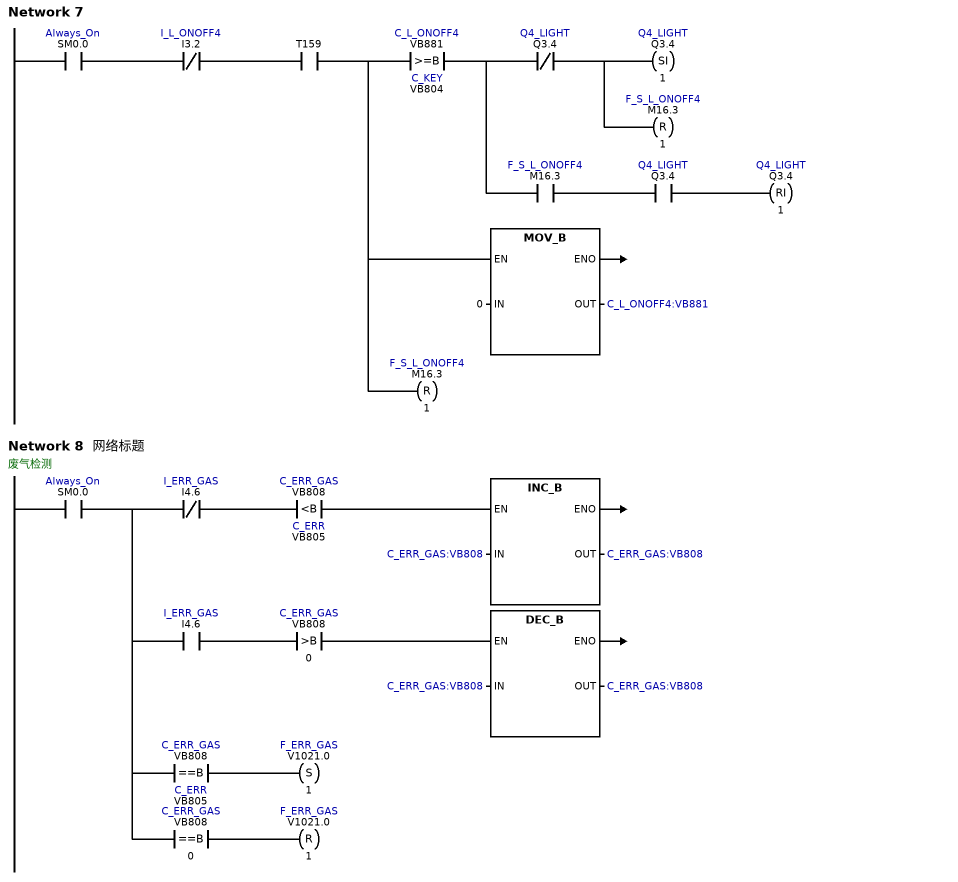
[picture p24: SBR3 networks 7-8]
Network 7
LD     Always_On:SM0.0
AN     I_L_ONOFF4:I3.2
A      T159
LPS
AB>=   C_L_ONOFF4:VB881, C_KEY:VB804
LPS
AN     Q4_LIGHT:Q3.4
SI     Q4_LIGHT:Q3.4, 1
R      F_S_L_ONOFF4:M16.3, 1
LPP
A      F_S_L_ONOFF4:M16.3
A      Q4_LIGHT:Q3.4
RI     Q4_LIGHT:Q3.4, 1
LPP
MOVB   0, C_L_ONOFF4:VB881
R      F_S_L_ONOFF4:M16.3, 1
Network 8 // 网络标题
// 废气检测
LD     Always_On:SM0.0
LPS
AN     I_ERR_GAS:I4.6
AB<    C_ERR_GAS:VB808, C_ERR:VB805
INCB   C_ERR_GAS:VB808
LRD
A      I_ERR_GAS:I4.6
AB>    C_ERR_GAS:VB808, 0
DECB   C_ERR_GAS:VB808
LRD
AB=    C_ERR_GAS:VB808, C_ERR:VB805
S      F_ERR_GAS:V1021.0, 1
LPP
AB=    C_ERR_GAS:VB808, 0
R      F_ERR_GAS:V1021.0, 1
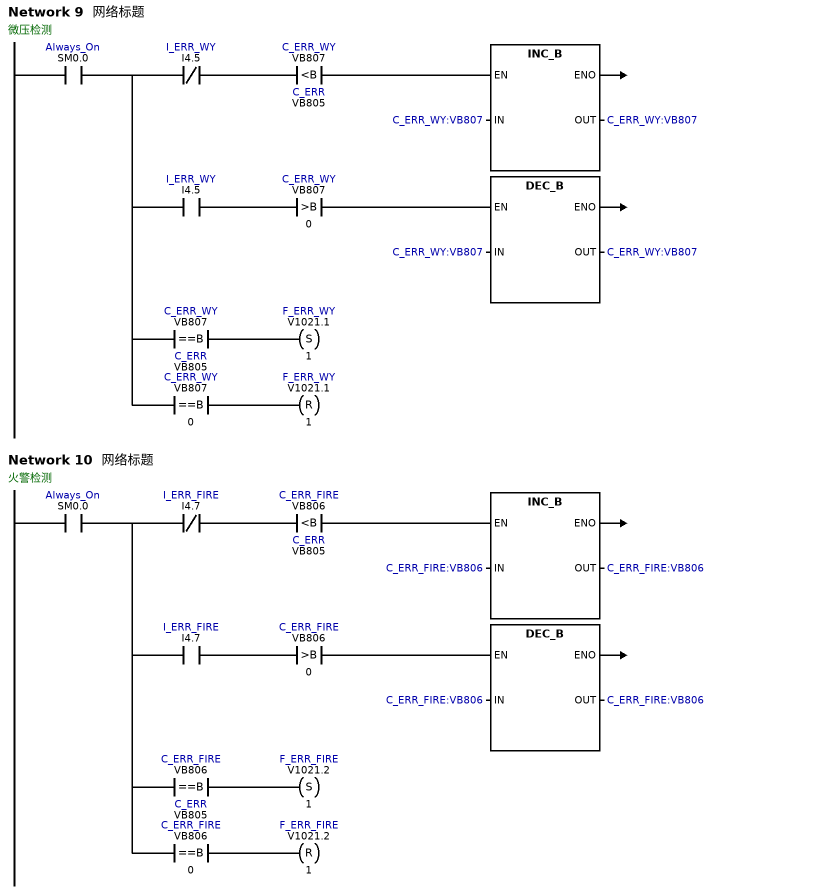
Network 9 // 网络标题
// 微压检测
LD     Always_On:SM0.0
LPS
AN     I_ERR_WY:I4.5
AB<    C_ERR_WY:VB807, C_ERR:VB805
INCB   C_ERR_WY:VB807
LRD
A      I_ERR_WY:I4.5
AB>    C_ERR_WY:VB807, 0
DECB   C_ERR_WY:VB807
LRD
AB=    C_ERR_WY:VB807, C_ERR:VB805
S      F_ERR_WY:V1021.1, 1
LPP
AB=    C_ERR_WY:VB807, 0
R      F_ERR_WY:V1021.1, 1
Network 10 // 网络标题
// 火警检测
LD     Always_On:SM0.0
LPS
AN     I_ERR_FIRE:I4.7
AB<    C_ERR_FIRE:VB806, C_ERR:VB805
INCB   C_ERR_FIRE:VB806
LRD
A      I_ERR_FIRE:I4.7
AB>    C_ERR_FIRE:VB806, 0
DECB   C_ERR_FIRE:VB806
LRD
AB=    C_ERR_FIRE:VB806, C_ERR:VB805
S      F_ERR_FIRE:V1021.2, 1
LPP
AB=    C_ERR_FIRE:VB806, 0
R      F_ERR_FIRE:V1021.2, 1
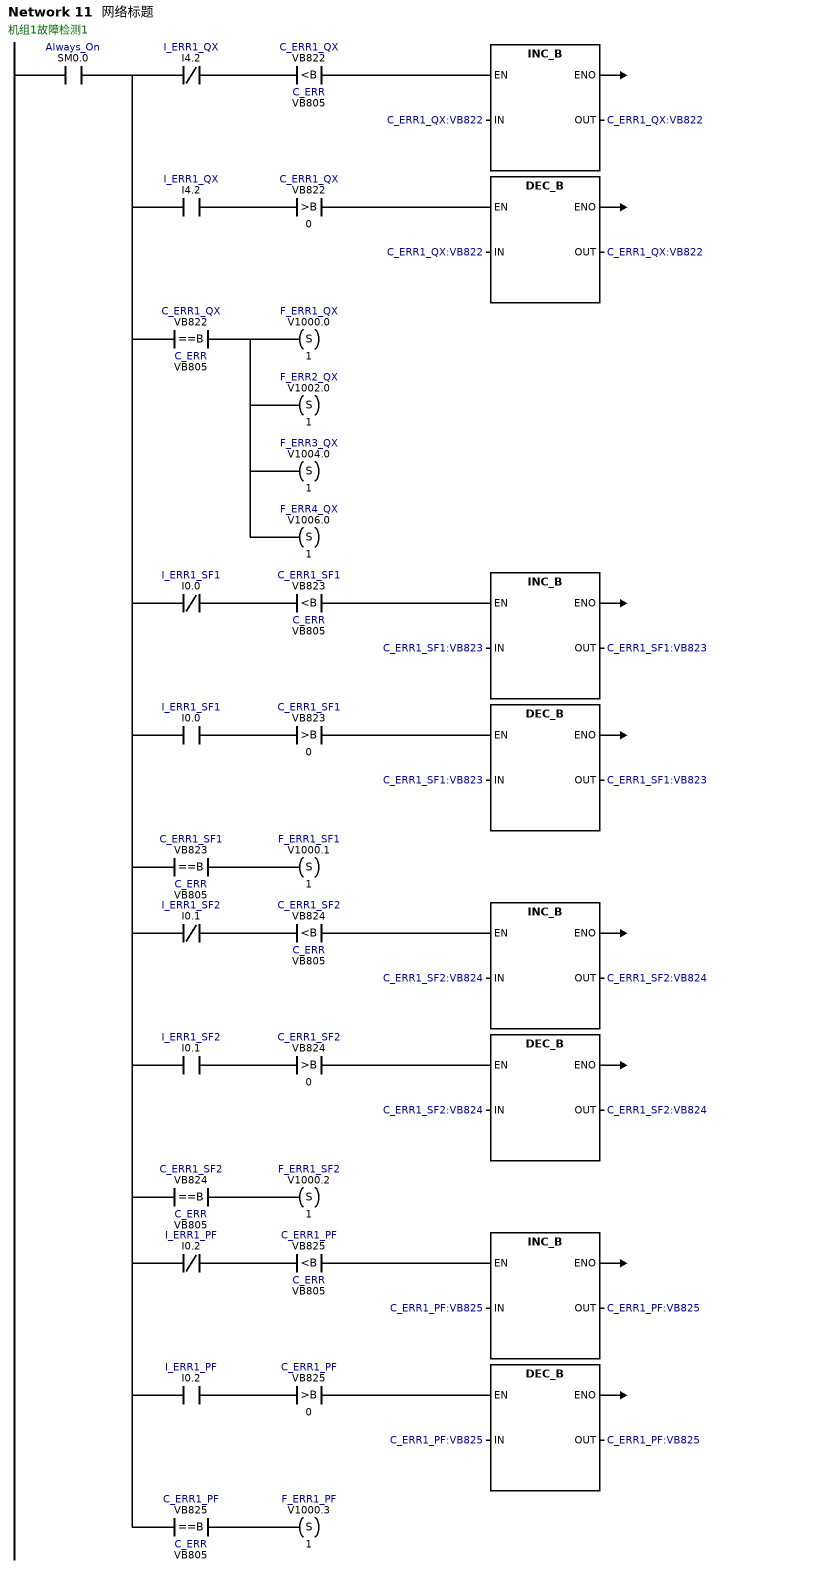
Network 11 // 网络标题
// 机组1故障检测1
LD     Always_On:SM0.0
LPS
AN     I_ERR1_QX:I4.2
AB<    C_ERR1_QX:VB822, C_ERR:VB805
INCB   C_ERR1_QX:VB822
LRD
A      I_ERR1_QX:I4.2
AB>    C_ERR1_QX:VB822, 0
DECB   C_ERR1_QX:VB822
LRD
AB=    C_ERR1_QX:VB822, C_ERR:VB805
S      F_ERR1_QX:V1000.0, 1
S      F_ERR2_QX:V1002.0, 1
S      F_ERR3_QX:V1004.0, 1
S      F_ERR4_QX:V1006.0, 1
LPP
LPS
AN     I_ERR1_SF1:I0.0
AB<    C_ERR1_SF1:VB823, C_ERR:VB805
INCB   C_ERR1_SF1:VB823
LRD
A      I_ERR1_SF1:I0.0
AB>    C_ERR1_SF1:VB823, 0
DECB   C_ERR1_SF1:VB823
LRD
AB=    C_ERR1_SF1:VB823, C_ERR:VB805
S      F_ERR1_SF1:V1000.1, 1
LRD
AN     I_ERR1_SF2:I0.1
AB<    C_ERR1_SF2:VB824, C_ERR:VB805
INCB   C_ERR1_SF2:VB824
LRD
A      I_ERR1_SF2:I0.1
AB>    C_ERR1_SF2:VB824, 0
DECB   C_ERR1_SF2:VB824
LRD
AB=    C_ERR1_SF2:VB824, C_ERR:VB805
S      F_ERR1_SF2:V1000.2, 1
LRD
AN     I_ERR1_PF:I0.2
AB<    C_ERR1_PF:VB825, C_ERR:VB805
INCB   C_ERR1_PF:VB825
LRD
A      I_ERR1_PF:I0.2
AB>    C_ERR1_PF:VB825, 0
DECB   C_ERR1_PF:VB825
LPP
AB=    C_ERR1_PF:VB825, C_ERR:VB805
S      F_ERR1_PF:V1000.3, 1
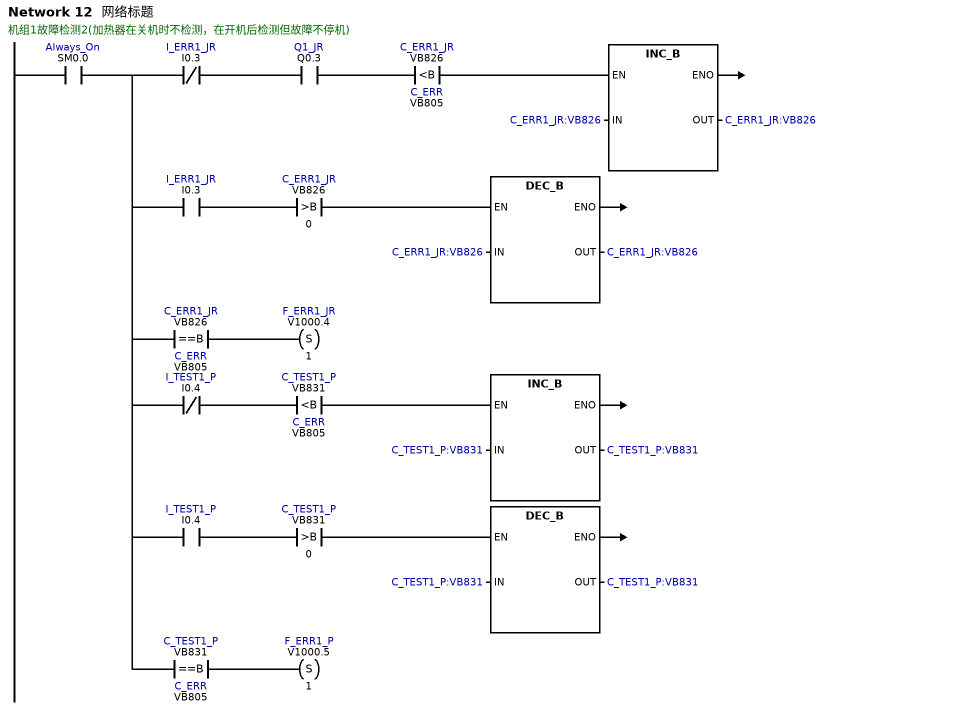
Network 12 // 网络标题
// 机组1故障检测2(加热器在关机时不检测，在开机后检测但故障不停机)
LD     Always_On:SM0.0
LPS
AN     I_ERR1_JR:I0.3
A      Q1_JR:Q0.3
AB<    C_ERR1_JR:VB826, C_ERR:VB805
INCB   C_ERR1_JR:VB826
LRD
A      I_ERR1_JR:I0.3
AB>    C_ERR1_JR:VB826, 0
DECB   C_ERR1_JR:VB826
LRD
AB=    C_ERR1_JR:VB826, C_ERR:VB805
S      F_ERR1_JR:V1000.4, 1
LRD
AN     I_TEST1_P:I0.4
AB<    C_TEST1_P:VB831, C_ERR:VB805
INCB   C_TEST1_P:VB831
LRD
A      I_TEST1_P:I0.4
AB>    C_TEST1_P:VB831, 0
DECB   C_TEST1_P:VB831
LPP
AB=    C_TEST1_P:VB831, C_ERR:VB805
S      F_ERR1_P:V1000.5, 1
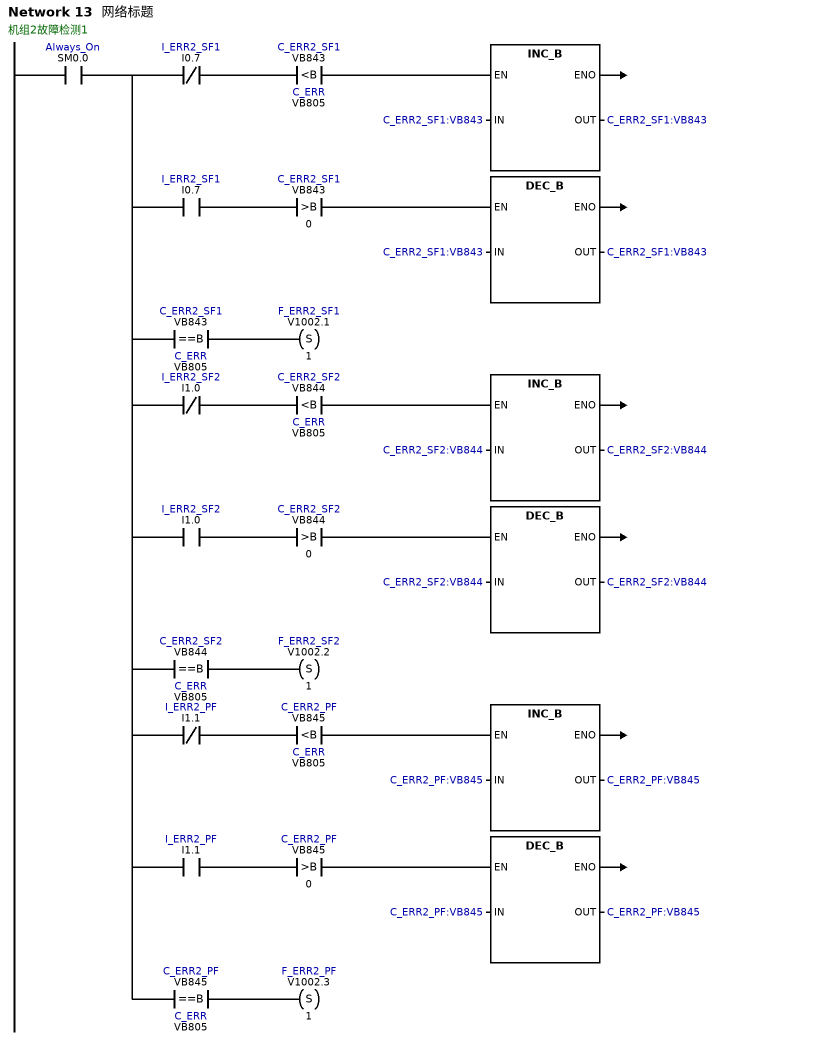
Network 13 // 网络标题
// 机组2故障检测1
LD     Always_On:SM0.0
LPS
AN     I_ERR2_SF1:I0.7
AB<    C_ERR2_SF1:VB843, C_ERR:VB805
INCB   C_ERR2_SF1:VB843
LRD
A      I_ERR2_SF1:I0.7
AB>    C_ERR2_SF1:VB843, 0
DECB   C_ERR2_SF1:VB843
LRD
AB=    C_ERR2_SF1:VB843, C_ERR:VB805
S      F_ERR2_SF1:V1002.1, 1
LRD
AN     I_ERR2_SF2:I1.0
AB<    C_ERR2_SF2:VB844, C_ERR:VB805
INCB   C_ERR2_SF2:VB844
LRD
A      I_ERR2_SF2:I1.0
AB>    C_ERR2_SF2:VB844, 0
DECB   C_ERR2_SF2:VB844
LRD
AB=    C_ERR2_SF2:VB844, C_ERR:VB805
S      F_ERR2_SF2:V1002.2, 1
LRD
AN     I_ERR2_PF:I1.1
AB<    C_ERR2_PF:VB845, C_ERR:VB805
INCB   C_ERR2_PF:VB845
LRD
A      I_ERR2_PF:I1.1
AB>    C_ERR2_PF:VB845, 0
DECB   C_ERR2_PF:VB845
LPP
AB=    C_ERR2_PF:VB845, C_ERR:VB805
S      F_ERR2_PF:V1002.3, 1
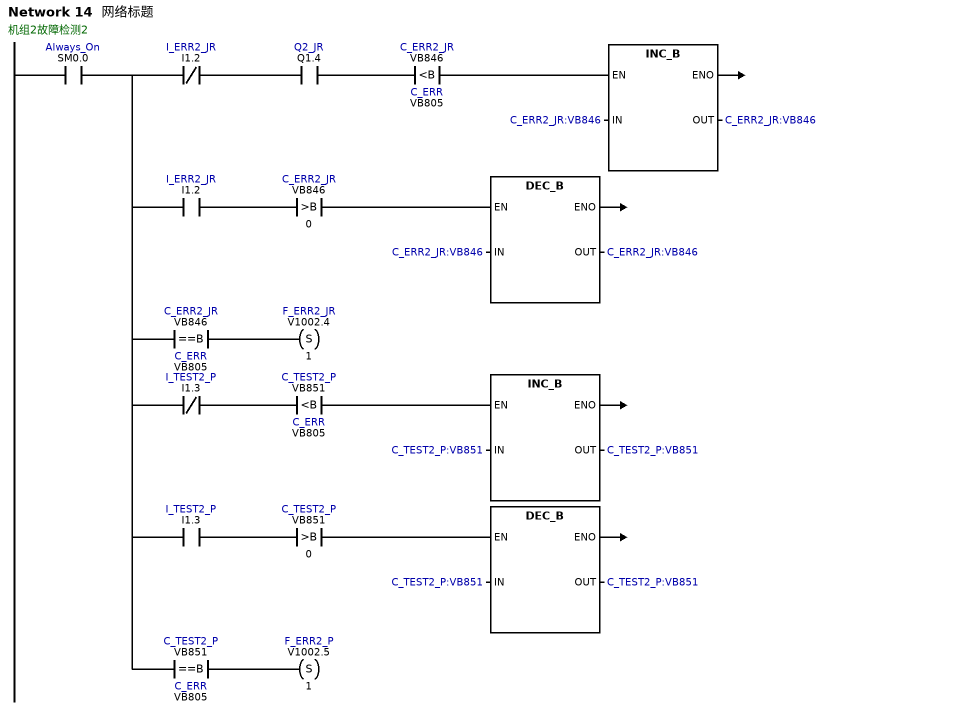
Network 14 // 网络标题
// 机组2故障检测2
LD     Always_On:SM0.0
LPS
AN     I_ERR2_JR:I1.2
A      Q2_JR:Q1.4
AB<    C_ERR2_JR:VB846, C_ERR:VB805
INCB   C_ERR2_JR:VB846
LRD
A      I_ERR2_JR:I1.2
AB>    C_ERR2_JR:VB846, 0
DECB   C_ERR2_JR:VB846
LRD
AB=    C_ERR2_JR:VB846, C_ERR:VB805
S      F_ERR2_JR:V1002.4, 1
LRD
AN     I_TEST2_P:I1.3
AB<    C_TEST2_P:VB851, C_ERR:VB805
INCB   C_TEST2_P:VB851
LRD
A      I_TEST2_P:I1.3
AB>    C_TEST2_P:VB851, 0
DECB   C_TEST2_P:VB851
LPP
AB=    C_TEST2_P:VB851, C_ERR:VB805
S      F_ERR2_P:V1002.5, 1
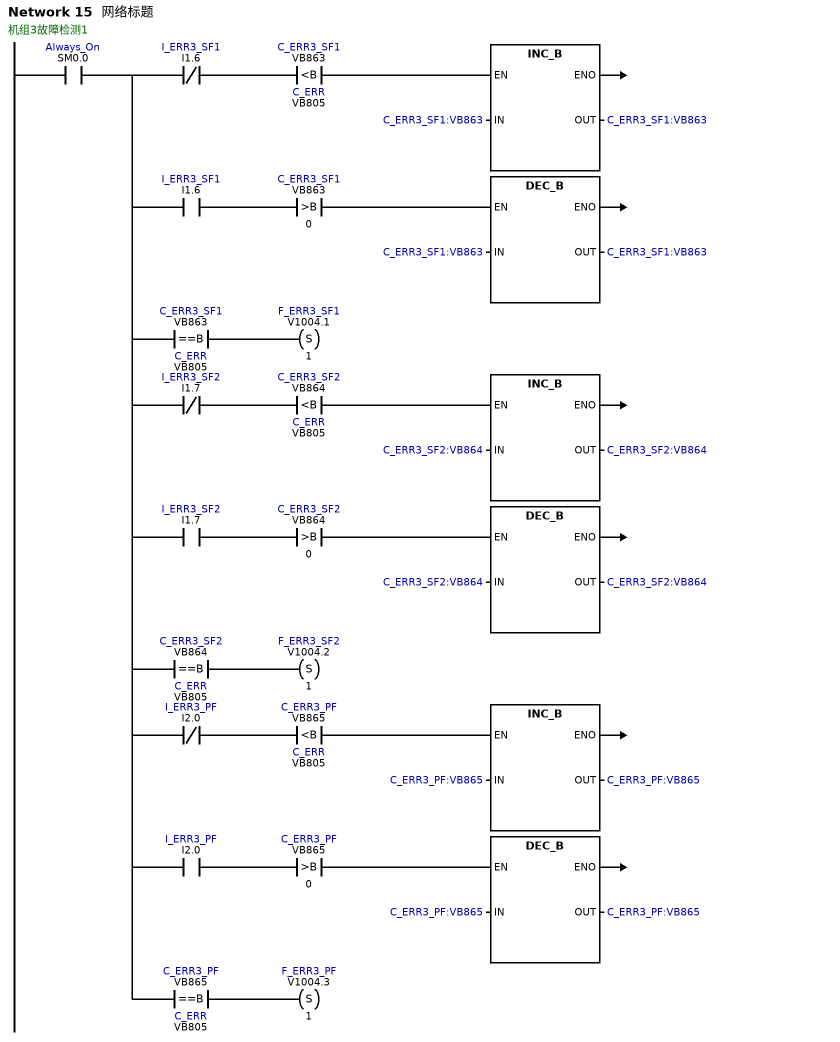
Network 15 // 网络标题
// 机组3故障检测1
LD     Always_On:SM0.0
LPS
AN     I_ERR3_SF1:I1.6
AB<    C_ERR3_SF1:VB863, C_ERR:VB805
INCB   C_ERR3_SF1:VB863
LRD
A      I_ERR3_SF1:I1.6
AB>    C_ERR3_SF1:VB863, 0
DECB   C_ERR3_SF1:VB863
LRD
AB=    C_ERR3_SF1:VB863, C_ERR:VB805
S      F_ERR3_SF1:V1004.1, 1
LRD
AN     I_ERR3_SF2:I1.7
AB<    C_ERR3_SF2:VB864, C_ERR:VB805
INCB   C_ERR3_SF2:VB864
LRD
A      I_ERR3_SF2:I1.7
AB>    C_ERR3_SF2:VB864, 0
DECB   C_ERR3_SF2:VB864
LRD
AB=    C_ERR3_SF2:VB864, C_ERR:VB805
S      F_ERR3_SF2:V1004.2, 1
LRD
AN     I_ERR3_PF:I2.0
AB<    C_ERR3_PF:VB865, C_ERR:VB805
INCB   C_ERR3_PF:VB865
LRD
A      I_ERR3_PF:I2.0
AB>    C_ERR3_PF:VB865, 0
DECB   C_ERR3_PF:VB865
LPP
AB=    C_ERR3_PF:VB865, C_ERR:VB805
S      F_ERR3_PF:V1004.3, 1
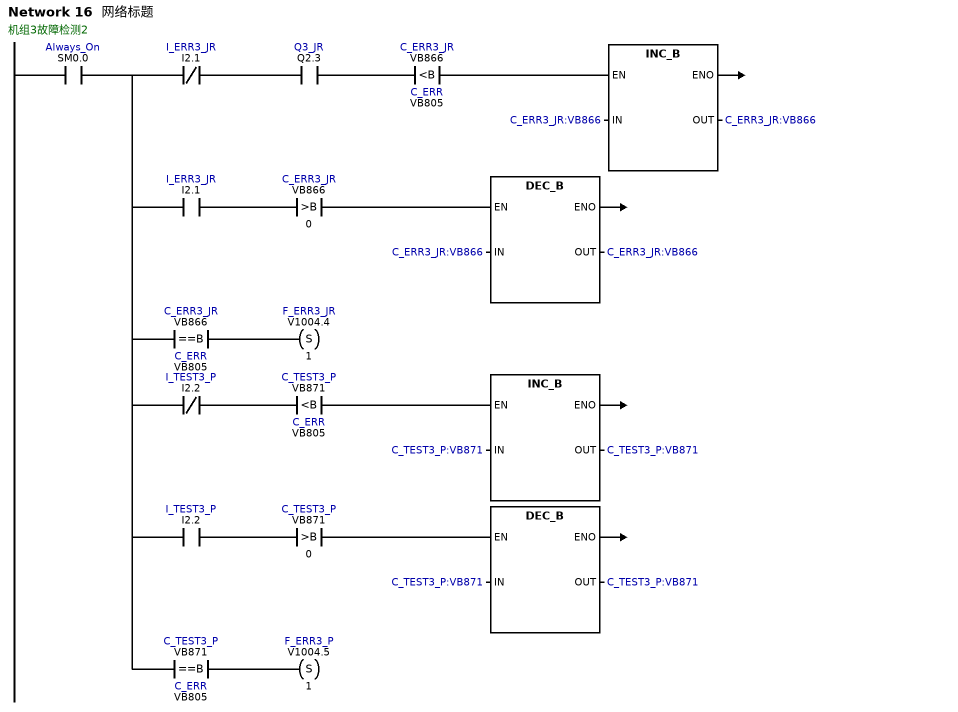
Network 16 // 网络标题
// 机组3故障检测2
LD     Always_On:SM0.0
LPS
AN     I_ERR3_JR:I2.1
A      Q3_JR:Q2.3
AB<    C_ERR3_JR:VB866, C_ERR:VB805
INCB   C_ERR3_JR:VB866
LRD
A      I_ERR3_JR:I2.1
AB>    C_ERR3_JR:VB866, 0
DECB   C_ERR3_JR:VB866
LRD
AB=    C_ERR3_JR:VB866, C_ERR:VB805
S      F_ERR3_JR:V1004.4, 1
LRD
AN     I_TEST3_P:I2.2
AB<    C_TEST3_P:VB871, C_ERR:VB805
INCB   C_TEST3_P:VB871
LRD
A      I_TEST3_P:I2.2
AB>    C_TEST3_P:VB871, 0
DECB   C_TEST3_P:VB871
LPP
AB=    C_TEST3_P:VB871, C_ERR:VB805
S      F_ERR3_P:V1004.5, 1
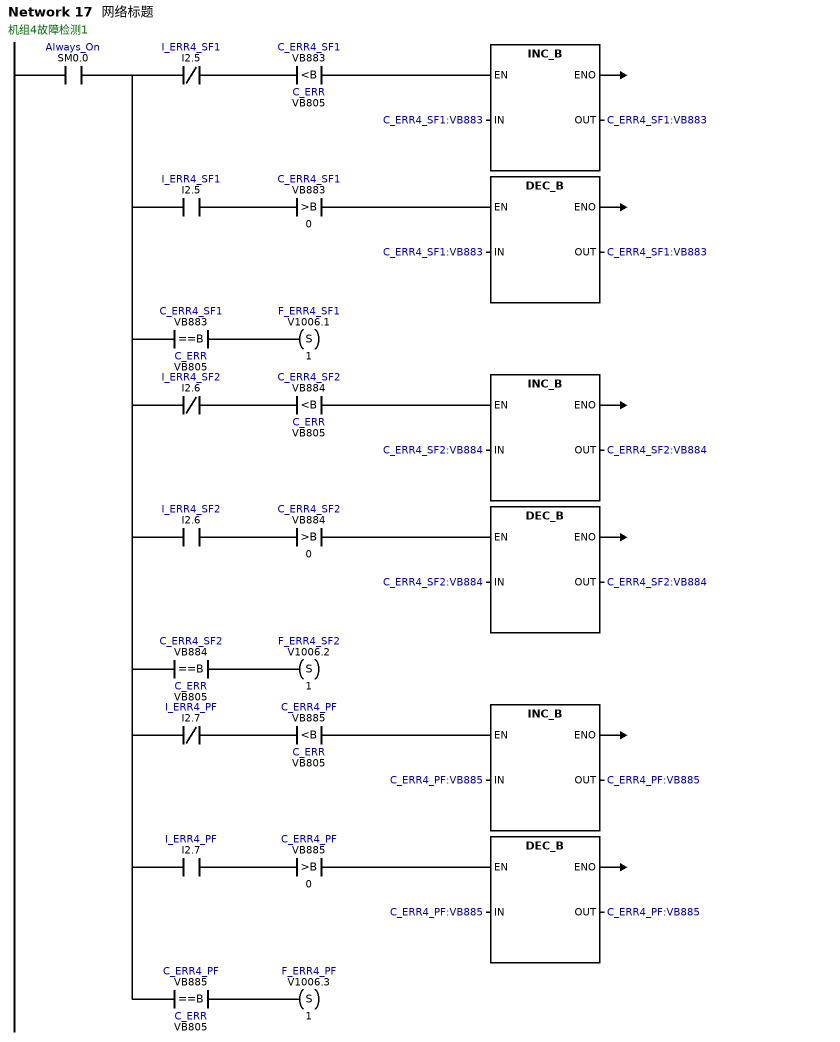
Network 17 // 网络标题
// 机组4故障检测1
LD     Always_On:SM0.0
LPS
AN     I_ERR4_SF1:I2.5
AB<    C_ERR4_SF1:VB883, C_ERR:VB805
INCB   C_ERR4_SF1:VB883
LRD
A      I_ERR4_SF1:I2.5
AB>    C_ERR4_SF1:VB883, 0
DECB   C_ERR4_SF1:VB883
LRD
AB=    C_ERR4_SF1:VB883, C_ERR:VB805
S      F_ERR4_SF1:V1006.1, 1
LRD
AN     I_ERR4_SF2:I2.6
AB<    C_ERR4_SF2:VB884, C_ERR:VB805
INCB   C_ERR4_SF2:VB884
LRD
A      I_ERR4_SF2:I2.6
AB>    C_ERR4_SF2:VB884, 0
DECB   C_ERR4_SF2:VB884
LRD
AB=    C_ERR4_SF2:VB884, C_ERR:VB805
S      F_ERR4_SF2:V1006.2, 1
LRD
AN     I_ERR4_PF:I2.7
AB<    C_ERR4_PF:VB885, C_ERR:VB805
INCB   C_ERR4_PF:VB885
LRD
A      I_ERR4_PF:I2.7
AB>    C_ERR4_PF:VB885, 0
DECB   C_ERR4_PF:VB885
LPP
AB=    C_ERR4_PF:VB885, C_ERR:VB805
S      F_ERR4_PF:V1006.3, 1
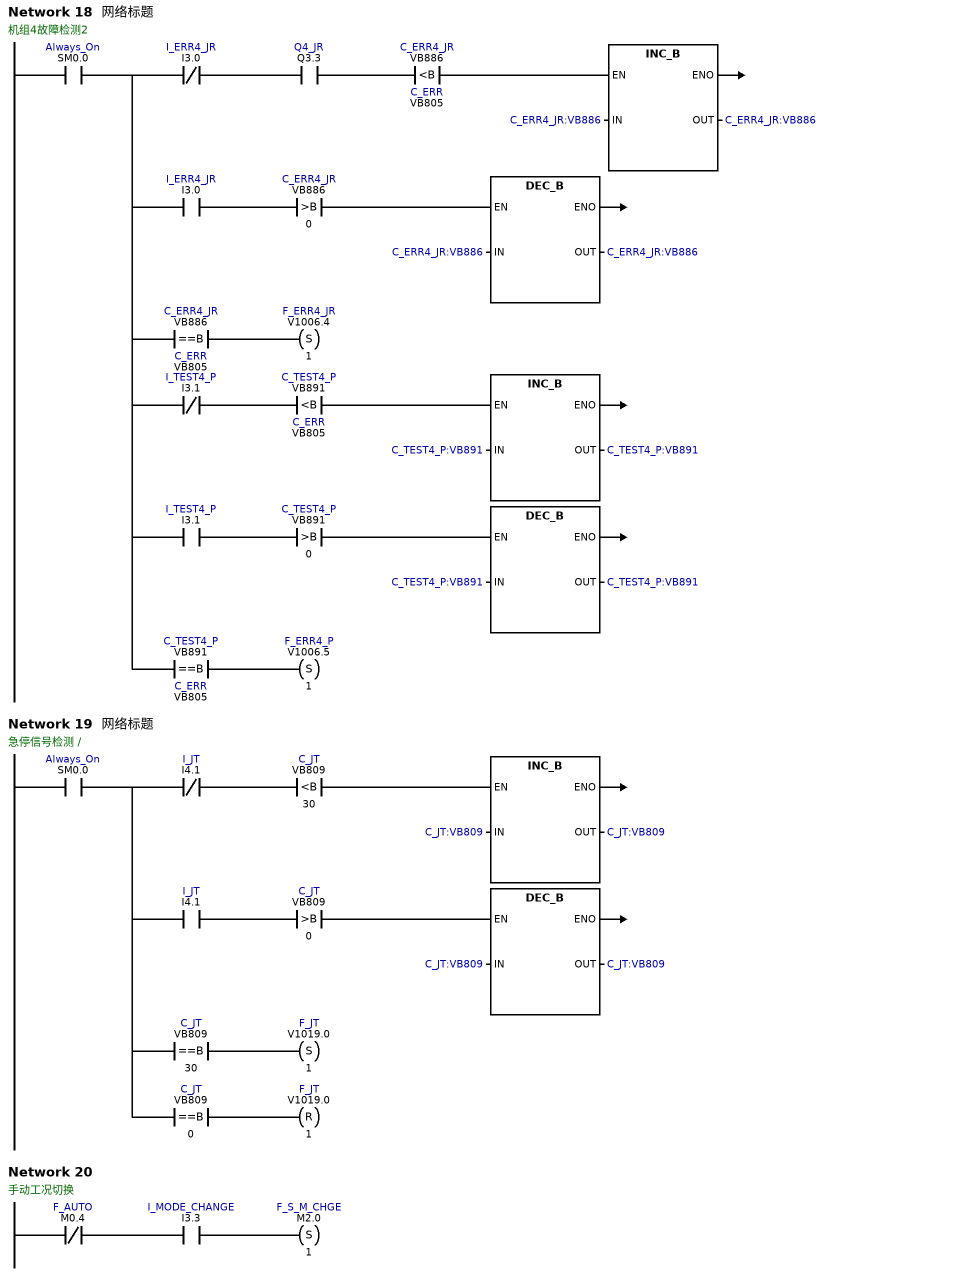
Network 18 // 网络标题
// 机组4故障检测2
LD     Always_On:SM0.0
LPS
AN     I_ERR4_JR:I3.0
A      Q4_JR:Q3.3
AB<    C_ERR4_JR:VB886, C_ERR:VB805
INCB   C_ERR4_JR:VB886
LRD
A      I_ERR4_JR:I3.0
AB>    C_ERR4_JR:VB886, 0
DECB   C_ERR4_JR:VB886
LRD
AB=    C_ERR4_JR:VB886, C_ERR:VB805
S      F_ERR4_JR:V1006.4, 1
LRD
AN     I_TEST4_P:I3.1
AB<    C_TEST4_P:VB891, C_ERR:VB805
INCB   C_TEST4_P:VB891
LRD
A      I_TEST4_P:I3.1
AB>    C_TEST4_P:VB891, 0
DECB   C_TEST4_P:VB891
LPP
AB=    C_TEST4_P:VB891, C_ERR:VB805
S      F_ERR4_P:V1006.5, 1
Network 19 // 网络标题
// 急停信号检测
// 
LD     Always_On:SM0.0
LPS
AN     I_JT:I4.1
AB<    C_JT:VB809, 30
INCB   C_JT:VB809
LRD
A      I_JT:I4.1
AB>    C_JT:VB809, 0
DECB   C_JT:VB809
LRD
AB=    C_JT:VB809, 30
S      F_JT:V1019.0, 1
LPP
AB=    C_JT:VB809, 0
R      F_JT:V1019.0, 1
Network 20
// 手动工况切换
LDN    F_AUTO:M0.4
A      I_MODE_CHANGE:I3.3
S      F_S_M_CHGE:M2.0, 1
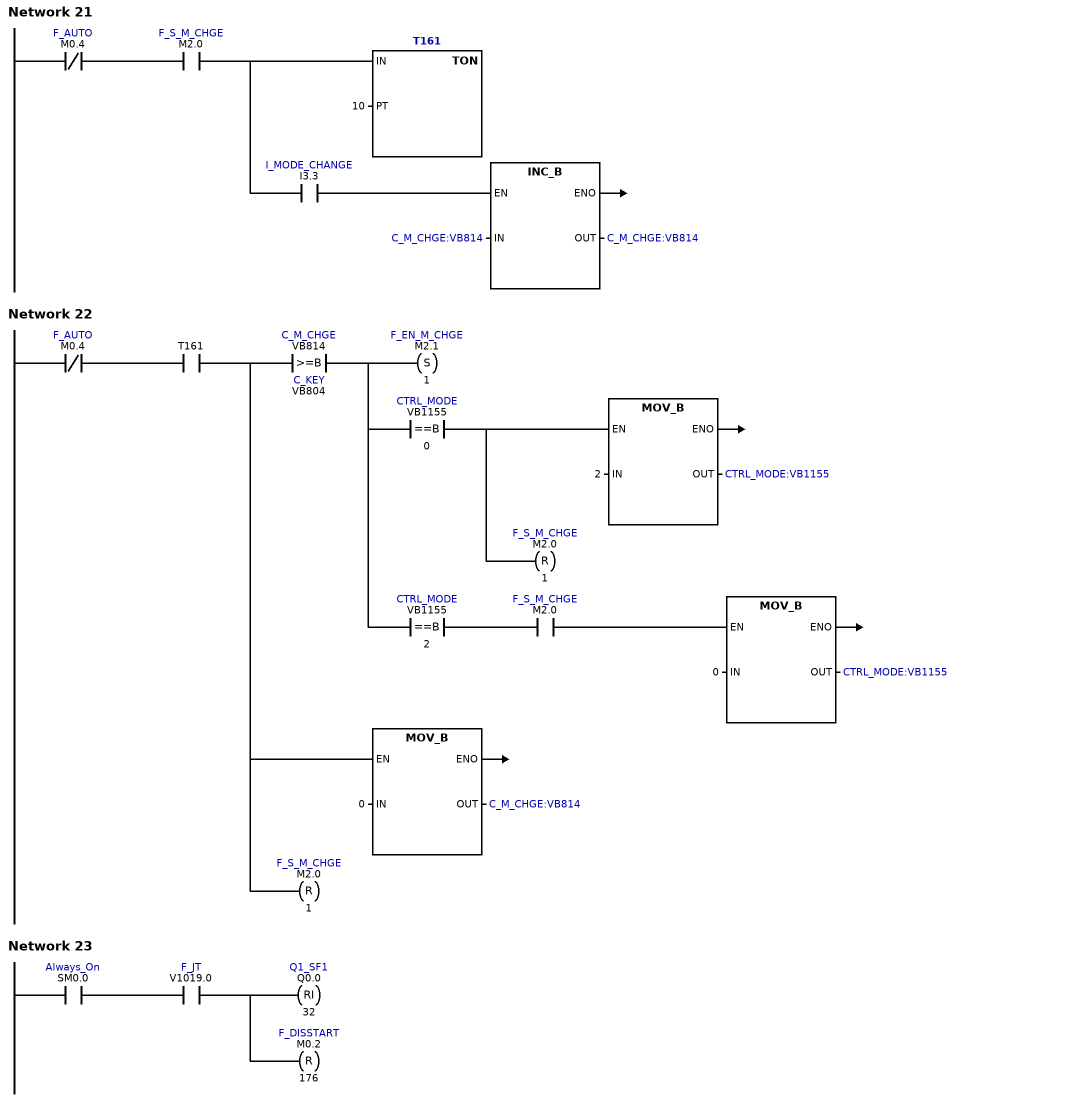
Network 21
LDN    F_AUTO:M0.4
A      F_S_M_CHGE:M2.0
TON    T161, 10
A      I_MODE_CHANGE:I3.3
INCB   C_M_CHGE:VB814
Network 22
LDN    F_AUTO:M0.4
A      T161
LPS
AB>=   C_M_CHGE:VB814, C_KEY:VB804
LPS
S      F_EN_M_CHGE:M2.1, 1
AB=    CTRL_MODE:VB1155, 0
MOVB   2, CTRL_MODE:VB1155
R      F_S_M_CHGE:M2.0, 1
LPP
AB=    CTRL_MODE:VB1155, 2
A      F_S_M_CHGE:M2.0
MOVB   0, CTRL_MODE:VB1155
LPP
MOVB   0, C_M_CHGE:VB814
R      F_S_M_CHGE:M2.0, 1
Network 23
LD     Always_On:SM0.0
A      F_JT:V1019.0
RI     Q1_SF1:Q0.0, 32
R      F_DISSTART:M0.2, 176
END_SUBROUTINE_BLOCK

SUBROUTINE_BLOCK HMI通讯参数:SBR4
TITLE=与HMI通讯有关参数更改
BEGIN
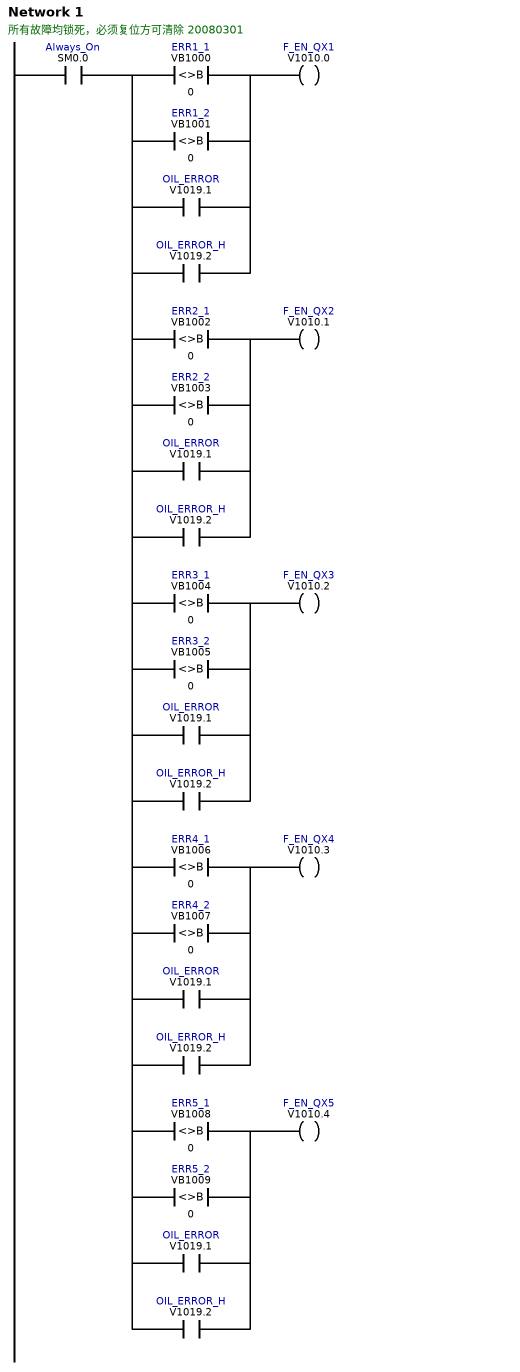
Network 1
// 所有故障均锁死，必须复位方可清除 20080301
// (network saved uncompiled; LAD cells follow)
// row 0: c0 -| |- Always_On:SM0.0 v  c1 -|<>B|- ERR1_1:VB1000, 0 v  c2 -( ) F_EN_QX1:V1010.0
// row 1: c0 ^v  c1 -|<>B|- ERR1_2:VB1001, 0 ^v
// row 2: c0 ^v  c1 -| |- OIL_ERROR:V1019.1 ^v
// row 3: c0 ^v  c1 -| |- OIL_ERROR_H:V1019.2 ^
// row 4: c0 ^v  c1 -|<>B|- ERR2_1:VB1002, 0 v  c2 -( ) F_EN_QX2:V1010.1
// row 5: c0 ^v  c1 -|<>B|- ERR2_2:VB1003, 0 ^v
// row 6: c0 ^v  c1 -| |- OIL_ERROR:V1019.1 ^v
// row 7: c0 ^v  c1 -| |- OIL_ERROR_H:V1019.2 ^
// row 8: c0 ^v  c1 -|<>B|- ERR3_1:VB1004, 0 v  c2 -( ) F_EN_QX3:V1010.2
// row 9: c0 ^v  c1 -|<>B|- ERR3_2:VB1005, 0 ^v
// row 10: c0 ^v  c1 -| |- OIL_ERROR:V1019.1 ^v
// row 11: c0 ^v  c1 -| |- OIL_ERROR_H:V1019.2 ^
// row 12: c0 ^v  c1 -|<>B|- ERR4_1:VB1006, 0 v  c2 -( ) F_EN_QX4:V1010.3
// row 13: c0 ^v  c1 -|<>B|- ERR4_2:VB1007, 0 ^v
// row 14: c0 ^v  c1 -| |- OIL_ERROR:V1019.1 ^v
// row 15: c0 ^v  c1 -| |- OIL_ERROR_H:V1019.2 ^
// row 16: c0 ^v  c1 -|<>B|- ERR5_1:VB1008, 0 v  c2 -( ) F_EN_QX5:V1010.4
// row 17: c0 ^v  c1 -|<>B|- ERR5_2:VB1009, 0 ^v
// row 18: c0 ^v  c1 -| |- OIL_ERROR:V1019.1 ^v
// row 19: c0 ^  c1 -| |- OIL_ERROR_H:V1019.2 ^
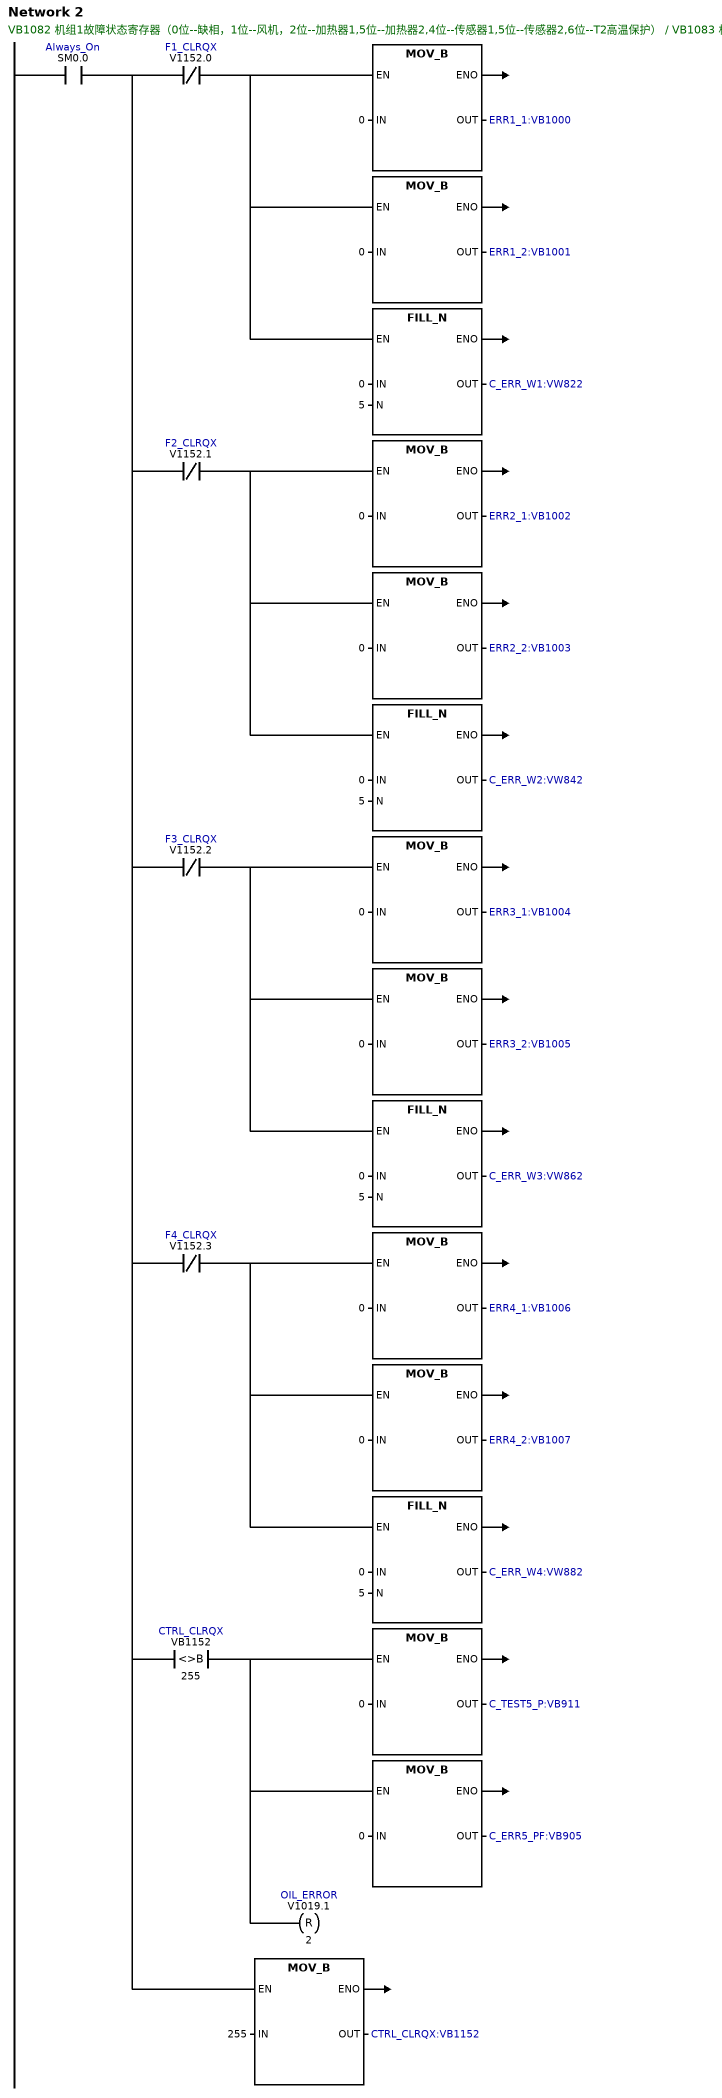
Network 2
// VB1082 机组1故障状态寄存器（0位--缺相，1位--风机，2位--加热器1,5位--加热器2,4位--传感器1,5位--传感器2,6位--T2高温保护）
// VB1083 机组2故障状态寄存器
// VB1084 机组3故障状态寄存器
// 复位所有故障
// (network saved uncompiled; LAD cells follow)
// row 0: c0 -| |- Always_On:SM0.0 v  c1 -|/|- F1_CLRQX:V1152.0 v  c2 --  c3 [MOV_B EN:=power@row0, IN:=0, ENO=>power, OUT=>ERR1_1:VB1000]  c4 ->
// row 1: c0 ^v  c1 ^v  c3 [box]
// row 2: c0 ^v  c1 ^v  c2 --  c3 [MOV_B EN:=power@row2, IN:=0, ENO=>power, OUT=>ERR1_2:VB1001]  c4 ->
// row 3: c0 ^v  c1 ^v  c3 [box]
// row 4: c0 ^v  c1 ^  c2 --  c3 [FILL_N EN:=power@row4, IN:=0, N:=5, ENO=>power, OUT=>C_ERR_W1:VW822]  c4 ->
// row 5: c0 ^v  c3 [box]
// row 6: c0 ^v  c1 -|/|- F2_CLRQX:V1152.1 v  c2 --  c3 [MOV_B EN:=power@row6, IN:=0, ENO=>power, OUT=>ERR2_1:VB1002]  c4 ->
// row 7: c0 ^v  c1 ^v  c3 [box]
// row 8: c0 ^v  c1 ^v  c2 --  c3 [MOV_B EN:=power@row8, IN:=0, ENO=>power, OUT=>ERR2_2:VB1003]  c4 ->
// row 9: c0 ^v  c1 ^v  c3 [box]
// row 10: c0 ^v  c1 ^  c2 --  c3 [FILL_N EN:=power@row10, IN:=0, N:=5, ENO=>power, OUT=>C_ERR_W2:VW842]  c4 ->
// row 11: c0 ^v  c3 [box]
// row 12: c0 ^v  c1 -|/|- F3_CLRQX:V1152.2 v  c2 --  c3 [MOV_B EN:=power@row12, IN:=0, ENO=>power, OUT=>ERR3_1:VB1004]  c4 ->
// row 13: c0 ^v  c1 ^v  c3 [box]
// row 14: c0 ^v  c1 ^v  c2 --  c3 [MOV_B EN:=power@row14, IN:=0, ENO=>power, OUT=>ERR3_2:VB1005]  c4 ->
// row 15: c0 ^v  c1 ^v  c3 [box]
// row 16: c0 ^v  c1 ^  c2 --  c3 [FILL_N EN:=power@row16, IN:=0, N:=5, ENO=>power, OUT=>C_ERR_W3:VW862]  c4 ->
// row 17: c0 ^v  c3 [box]
// row 18: c0 ^v  c1 -|/|- F4_CLRQX:V1152.3 v  c2 --  c3 [MOV_B EN:=power@row18, IN:=0, ENO=>power, OUT=>ERR4_1:VB1006]  c4 ->
// row 19: c0 ^v  c1 ^v  c3 [box]
// row 20: c0 ^v  c1 ^v  c2 --  c3 [MOV_B EN:=power@row20, IN:=0, ENO=>power, OUT=>ERR4_2:VB1007]  c4 ->
// row 21: c0 ^v  c1 ^v  c3 [box]
// row 22: c0 ^v  c1 ^  c2 --  c3 [FILL_N EN:=power@row22, IN:=0, N:=5, ENO=>power, OUT=>C_ERR_W4:VW882]  c4 ->
// row 23: c0 ^v  c3 [box]
// row 24: c0 ^v  c1 -|<>B|- CTRL_CLRQX:VB1152, 255 v  c2 --  c3 [MOV_B EN:=power@row24, IN:=0, ENO=>power, OUT=>C_TEST5_P:VB911]  c4 ->
// row 25: c0 ^v  c1 ^v  c3 [box]
// row 26: c0 ^v  c1 ^v  c2 --  c3 [MOV_B EN:=power@row26, IN:=0, ENO=>power, OUT=>C_ERR5_PF:VB905]  c4 ->
// row 27: c0 ^v  c1 ^v  c3 [box]
// row 28: c0 ^v  c1 ^  c2 -(R) OIL_ERROR:V1019.1, 2
// row 29: c0 ^  c1 --  c2 [MOV_B EN:=power@row29, IN:=255, ENO=>power, OUT=>CTRL_CLRQX:VB1152]  c3 ->
// row 30: c2 [box]
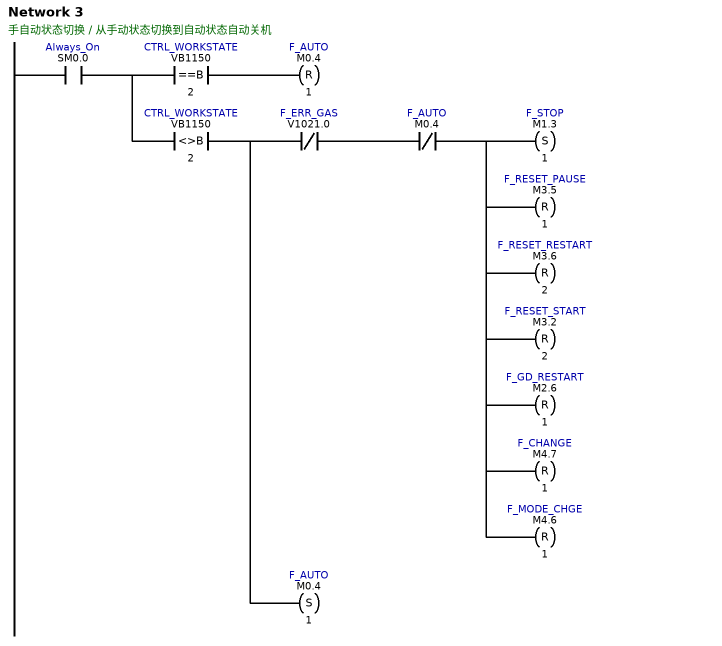
Network 3
// 手自动状态切换
// 从手动状态切换到自动状态自动关机
// (network saved uncompiled; LAD cells follow)
// row 0: c0 -| |- Always_On:SM0.0 v  c1 -|==B|- CTRL_WORKSTATE:VB1150, 2  c2 -(R) F_AUTO:M0.4, 1
// row 1: c0 ^  c1 -|<>B|- CTRL_WORKSTATE:VB1150, 2 v  c2 -|/|- F_ERR_GAS:V1021.0  c3 -|/|- F_AUTO:M0.4 v  c4 -(S) F_STOP:M1.3, 1
// row 2: c1 ^v  c3 ^v  c4 -(R) F_RESET_PAUSE:M3.5, 1
// row 3: c1 ^v  c3 ^v  c4 -(R) F_RESET_RESTART:M3.6, 2
// row 4: c1 ^v  c3 ^v  c4 -(R) F_RESET_START:M3.2, 2
// row 5: c1 ^v  c3 ^v  c4 -(R) F_GD_RESTART:M2.6, 1
// row 6: c1 ^v  c3 ^v  c4 -(R) F_CHANGE:M4.7, 1
// row 7: c1 ^v  c3 ^  c4 -(R) F_MODE_CHGE:M4.6, 1
// row 8: c1 ^  c2 -(S) F_AUTO:M0.4, 1
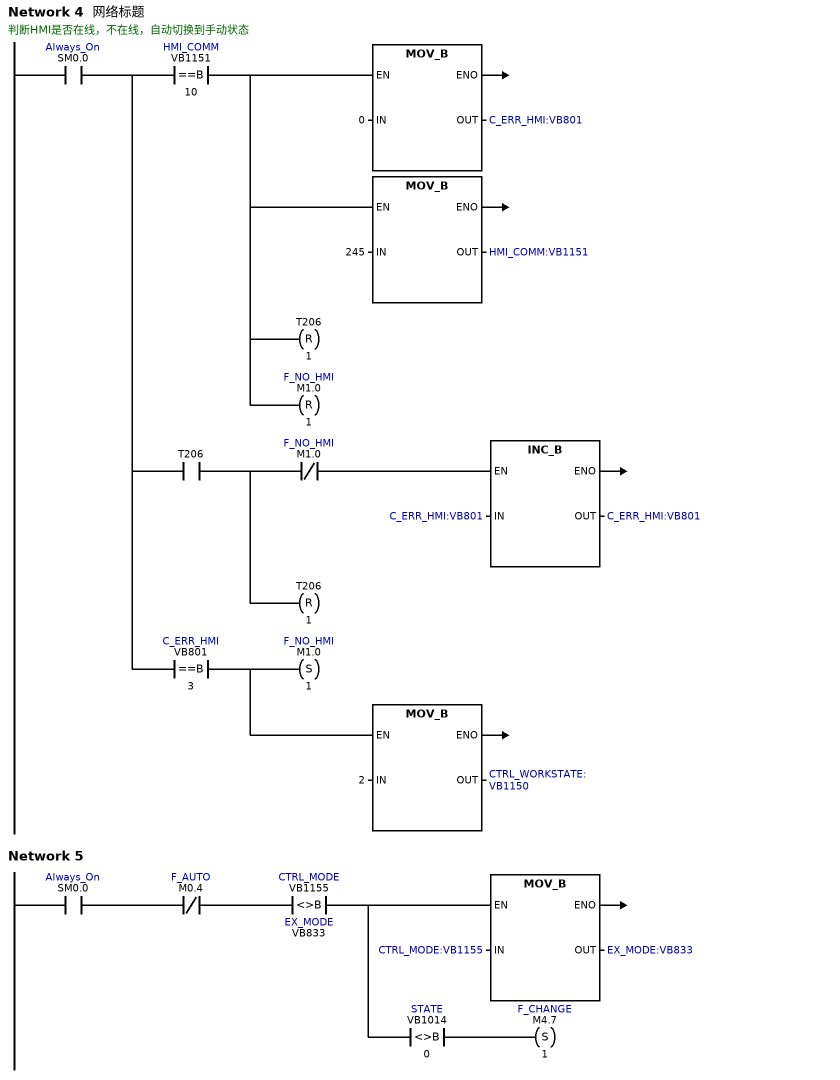
Network 4 // 网络标题
// 判断HMI是否在线，不在线，自动切换到手动状态
// (network saved uncompiled; LAD cells follow)
// row 0: c0 -| |- Always_On:SM0.0 v  c1 -|==B|- HMI_COMM:VB1151, 10 v  c2 --  c3 [MOV_B EN:=power@row0, IN:=0, ENO=>power, OUT=>C_ERR_HMI:VB801]  c4 ->
// row 1: c0 ^v  c1 ^v  c3 [box]
// row 2: c0 ^v  c1 ^v  c2 --  c3 [MOV_B EN:=power@row2, IN:=245, ENO=>power, OUT=>HMI_COMM:VB1151]  c4 ->
// row 3: c0 ^v  c1 ^v  c3 [box]
// row 4: c0 ^v  c1 ^v  c2 -(R) T206, 1
// row 5: c0 ^v  c1 ^  c2 -(R) F_NO_HMI:M1.0, 1
// row 6: c0 ^v  c1 -| |- T206 v  c2 -|/|- F_NO_HMI:M1.0  c3 --  c4 [INC_B EN:=power@row6, IN:=C_ERR_HMI:VB801, ENO=>power, OUT=>C_ERR_HMI:VB801]  c5 ->
// row 7: c0 ^v  c1 ^v  c4 [box]
// row 8: c0 ^v  c1 ^  c2 -(R) T206, 1
// row 9: c0 ^  c1 -|==B|- C_ERR_HMI:VB801, 3 v  c2 -(S) F_NO_HMI:M1.0, 1
// row 10: c1 ^  c2 --  c3 [MOV_B EN:=power@row10, IN:=2, ENO=>power, OUT=>CTRL_WORKSTATE:VB1150]  c4 ->
// row 11: c3 [box]
Network 5
// (network saved uncompiled; LAD cells follow)
// row 0: c0 -| |- Always_On:SM0.0  c1 -|/|- F_AUTO:M0.4  c2 -|<>B|- CTRL_MODE:VB1155, EX_MODE:VB833 v  c3 --  c4 [MOV_B EN:=power@row0, IN:=CTRL_MODE:VB1155, ENO=>power, OUT=>EX_MODE:VB833]  c5 ->
// row 1: c2 ^v  c4 [box]
// row 2: c2 ^  c3 -|<>B|- STATE:VB1014, 0  c4 -(S) F_CHANGE:M4.7, 1
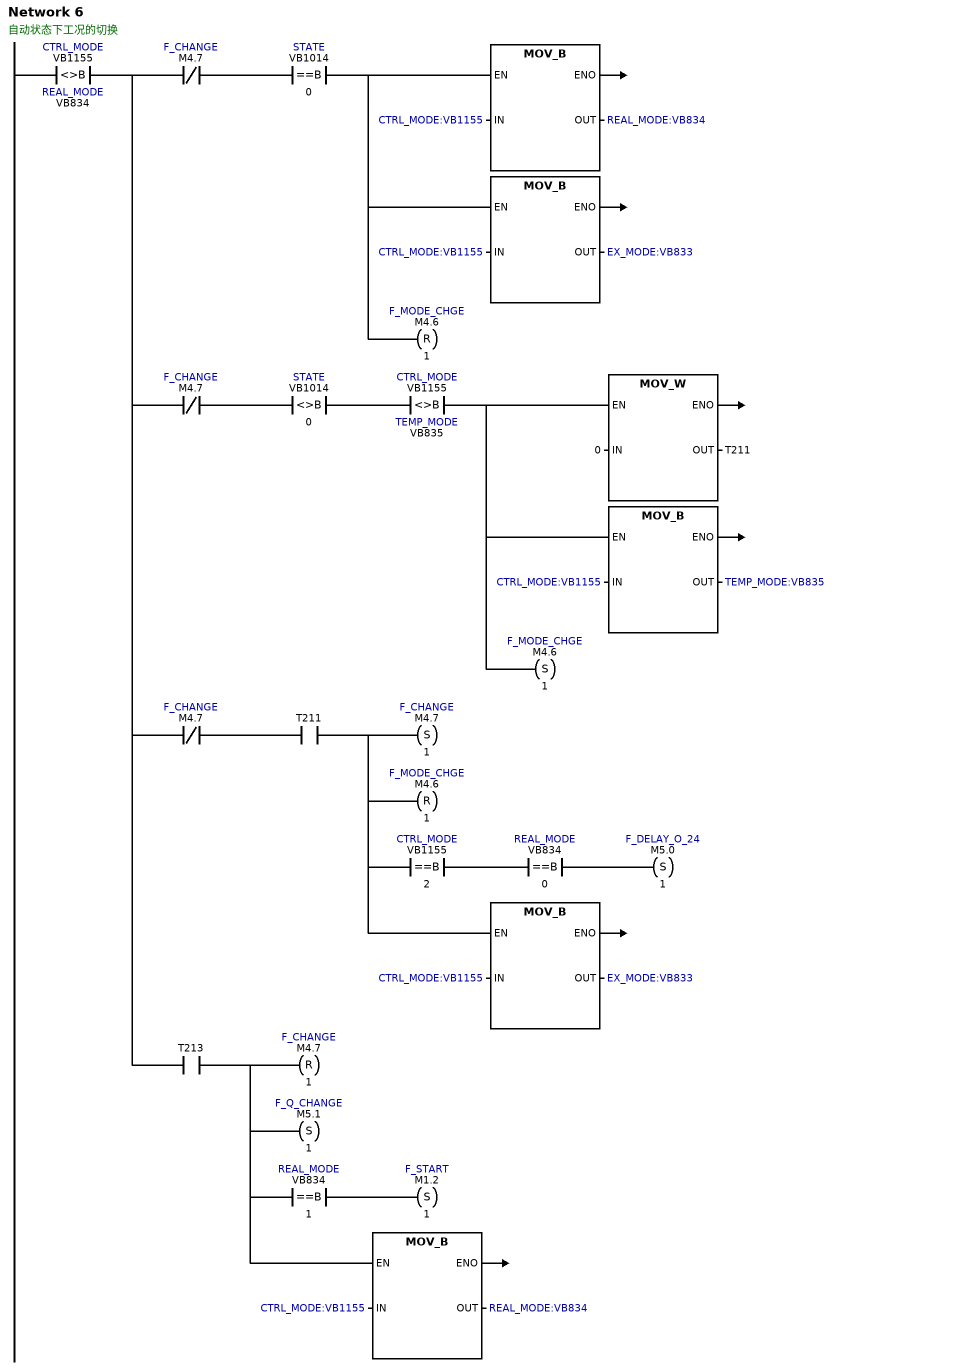
Network 6
// 自动状态下工况的切换
// (network saved uncompiled; LAD cells follow)
// row 0: c0 -|<>B|- CTRL_MODE:VB1155, REAL_MODE:VB834 v  c1 -|/|- F_CHANGE:M4.7  c2 -|==B|- STATE:VB1014, 0 v  c3 --  c4 [MOV_B EN:=power@row0, IN:=CTRL_MODE:VB1155, ENO=>power, OUT=>REAL_MODE:VB834]  c5 ->
// row 1: c0 ^v  c2 ^v  c4 [box]
// row 2: c0 ^v  c2 ^v  c3 --  c4 [MOV_B EN:=power@row2, IN:=CTRL_MODE:VB1155, ENO=>power, OUT=>EX_MODE:VB833]  c5 ->
// row 3: c0 ^v  c2 ^v  c4 [box]
// row 4: c0 ^v  c2 ^  c3 -(R) F_MODE_CHGE:M4.6, 1
// row 5: c0 ^v  c1 -|/|- F_CHANGE:M4.7  c2 -|<>B|- STATE:VB1014, 0  c3 -|<>B|- CTRL_MODE:VB1155, TEMP_MODE:VB835 v  c4 --  c5 [MOV_W EN:=power@row5, IN:=0, ENO=>power, OUT=>T211]  c6 ->
// row 6: c0 ^v  c3 ^v  c5 [box]
// row 7: c0 ^v  c3 ^v  c4 --  c5 [MOV_B EN:=power@row7, IN:=CTRL_MODE:VB1155, ENO=>power, OUT=>TEMP_MODE:VB835]  c6 ->
// row 8: c0 ^v  c3 ^v  c5 [box]
// row 9: c0 ^v  c3 ^  c4 -(S) F_MODE_CHGE:M4.6, 1
// row 10: c0 ^v  c1 -|/|- F_CHANGE:M4.7  c2 -| |- T211 v  c3 -(S) F_CHANGE:M4.7, 1
// row 11: c0 ^v  c2 ^v  c3 -(R) F_MODE_CHGE:M4.6, 1
// row 12: c0 ^v  c2 ^v  c3 -|==B|- CTRL_MODE:VB1155, 2  c4 -|==B|- REAL_MODE:VB834, 0  c5 -(S) F_DELAY_O_24:M5.0, 1
// row 13: c0 ^v  c2 ^  c3 --  c4 [MOV_B EN:=power@row13, IN:=CTRL_MODE:VB1155, ENO=>power, OUT=>EX_MODE:VB833]  c5 ->
// row 14: c0 ^v  c4 [box]
// row 15: c0 ^  c1 -| |- T213 v  c2 -(R) F_CHANGE:M4.7, 1
// row 16: c1 ^v  c2 -(S) F_Q_CHANGE:M5.1, 1
// row 17: c1 ^v  c2 -|==B|- REAL_MODE:VB834, 1  c3 -(S) F_START:M1.2, 1
// row 18: c1 ^  c2 --  c3 [MOV_B EN:=power@row18, IN:=CTRL_MODE:VB1155, ENO=>power, OUT=>REAL_MODE:VB834]  c4 ->
// row 19: c3 [box]
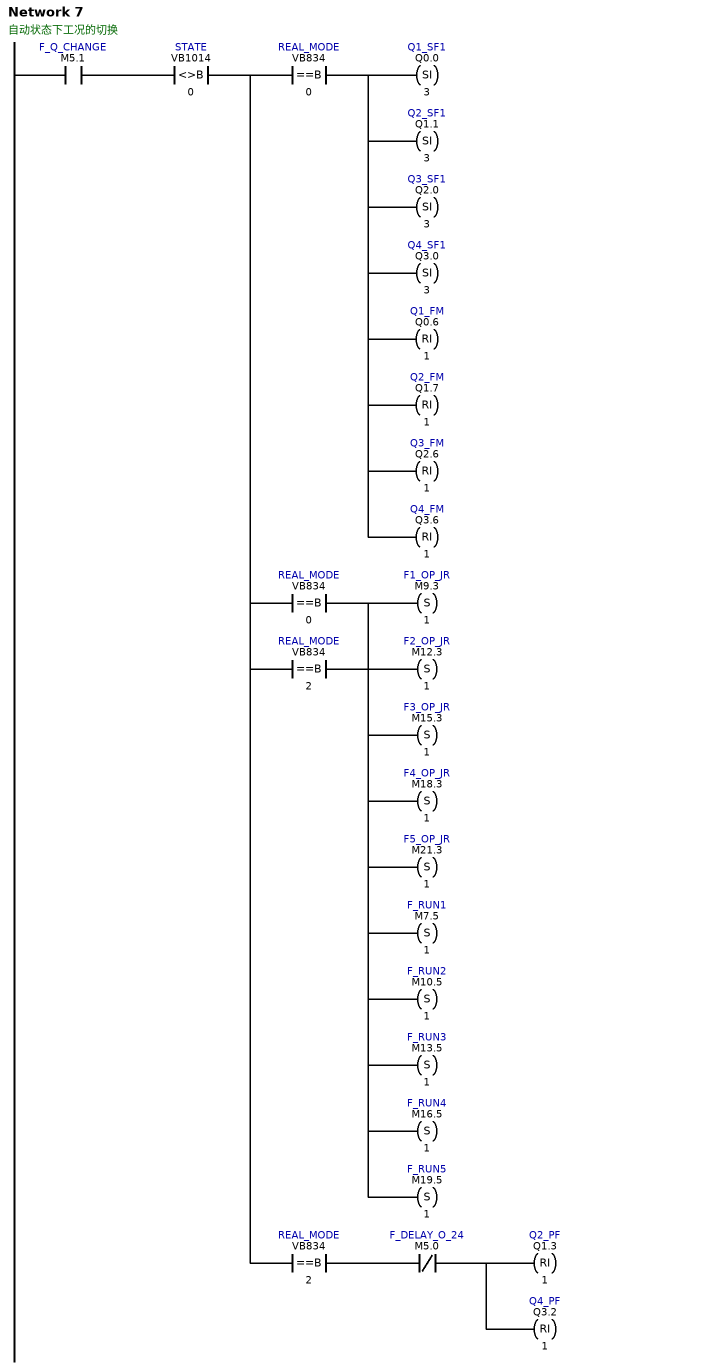
Network 7
// 自动状态下工况的切换
// (network saved uncompiled; LAD cells follow)
// row 0: c0 -| |- F_Q_CHANGE:M5.1  c1 -|<>B|- STATE:VB1014, 0 v  c2 -|==B|- REAL_MODE:VB834, 0 v  c3 -(SI) Q1_SF1:Q0.0, 3
// row 1: c1 ^v  c2 ^v  c3 -(SI) Q2_SF1:Q1.1, 3
// row 2: c1 ^v  c2 ^v  c3 -(SI) Q3_SF1:Q2.0, 3
// row 3: c1 ^v  c2 ^v  c3 -(SI) Q4_SF1:Q3.0, 3
// row 4: c1 ^v  c2 ^v  c3 -(RI) Q1_FM:Q0.6, 1
// row 5: c1 ^v  c2 ^v  c3 -(RI) Q2_FM:Q1.7, 1
// row 6: c1 ^v  c2 ^v  c3 -(RI) Q3_FM:Q2.6, 1
// row 7: c1 ^v  c2 ^  c3 -(RI) Q4_FM:Q3.6, 1
// row 8: c1 ^v  c2 -|==B|- REAL_MODE:VB834, 0 v  c3 -(S) F1_OP_JR:M9.3, 1
// row 9: c1 ^v  c2 -|==B|- REAL_MODE:VB834, 2 ^v  c3 -(S) F2_OP_JR:M12.3, 1
// row 10: c1 ^v  c2 ^v  c3 -(S) F3_OP_JR:M15.3, 1
// row 11: c1 ^v  c2 ^v  c3 -(S) F4_OP_JR:M18.3, 1
// row 12: c1 ^v  c2 ^v  c3 -(S) F5_OP_JR:M21.3, 1
// row 13: c1 ^v  c2 ^v  c3 -(S) F_RUN1:M7.5, 1
// row 14: c1 ^v  c2 ^v  c3 -(S) F_RUN2:M10.5, 1
// row 15: c1 ^v  c2 ^v  c3 -(S) F_RUN3:M13.5, 1
// row 16: c1 ^v  c2 ^v  c3 -(S) F_RUN4:M16.5, 1
// row 17: c1 ^v  c2 ^  c3 -(S) F_RUN5:M19.5, 1
// row 18: c1 ^  c2 -|==B|- REAL_MODE:VB834, 2  c3 -|/|- F_DELAY_O_24:M5.0 v  c4 -(RI) Q2_PF:Q1.3, 1
// row 19: c3 ^  c4 -(RI) Q4_PF:Q3.2, 1
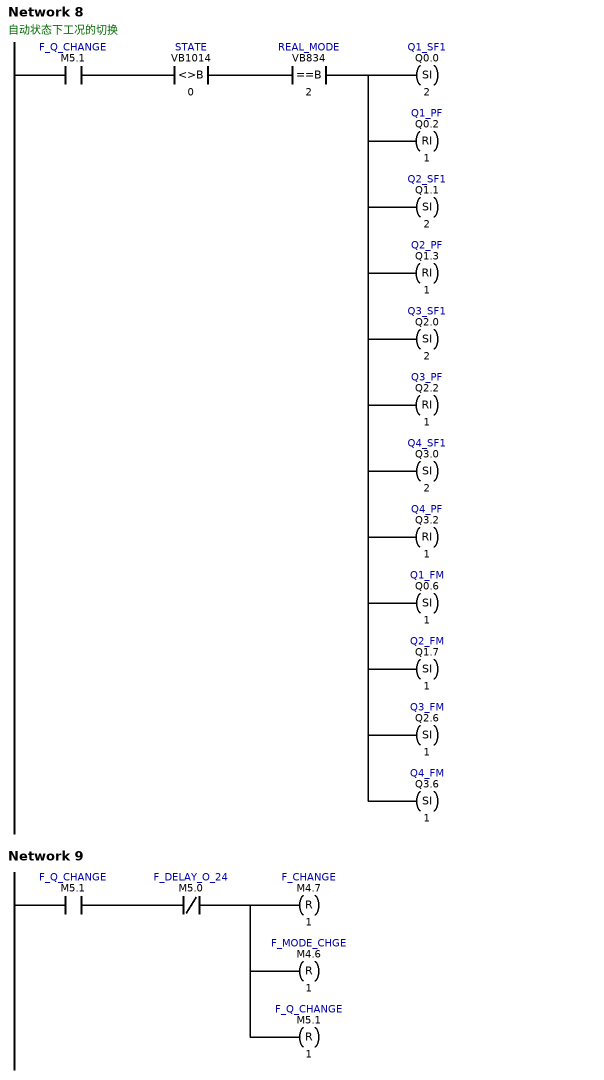
Network 8
// 自动状态下工况的切换
// (network saved uncompiled; LAD cells follow)
// row 0: c0 -| |- F_Q_CHANGE:M5.1  c1 -|<>B|- STATE:VB1014, 0  c2 -|==B|- REAL_MODE:VB834, 2 v  c3 -(SI) Q1_SF1:Q0.0, 2
// row 1: c2 ^v  c3 -(RI) Q1_PF:Q0.2, 1
// row 2: c2 ^v  c3 -(SI) Q2_SF1:Q1.1, 2
// row 3: c2 ^v  c3 -(RI) Q2_PF:Q1.3, 1
// row 4: c2 ^v  c3 -(SI) Q3_SF1:Q2.0, 2
// row 5: c2 ^v  c3 -(RI) Q3_PF:Q2.2, 1
// row 6: c2 ^v  c3 -(SI) Q4_SF1:Q3.0, 2
// row 7: c2 ^v  c3 -(RI) Q4_PF:Q3.2, 1
// row 8: c2 ^v  c3 -(SI) Q1_FM:Q0.6, 1
// row 9: c2 ^v  c3 -(SI) Q2_FM:Q1.7, 1
// row 10: c2 ^v  c3 -(SI) Q3_FM:Q2.6, 1
// row 11: c2 ^  c3 -(SI) Q4_FM:Q3.6, 1
Network 9
// (network saved uncompiled; LAD cells follow)
// row 0: c0 -| |- F_Q_CHANGE:M5.1  c1 -|/|- F_DELAY_O_24:M5.0 v  c2 -(R) F_CHANGE:M4.7, 1
// row 1: c1 ^v  c2 -(R) F_MODE_CHGE:M4.6, 1
// row 2: c1 ^  c2 -(R) F_Q_CHANGE:M5.1, 1
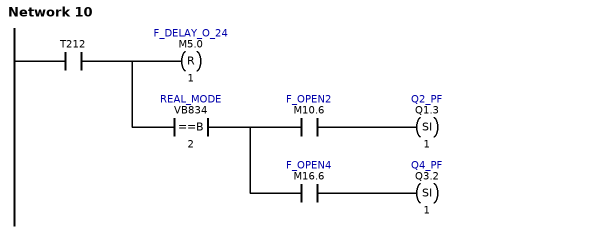
Network 10
// (network saved uncompiled; LAD cells follow)
// row 0: c0 -| |- T212 v  c1 -(R) F_DELAY_O_24:M5.0, 1
// row 1: c0 ^  c1 -|==B|- REAL_MODE:VB834, 2 v  c2 -| |- F_OPEN2:M10.6  c3 -(SI) Q2_PF:Q1.3, 1
// row 2: c1 ^  c2 -| |- F_OPEN4:M16.6  c3 -(SI) Q4_PF:Q3.2, 1
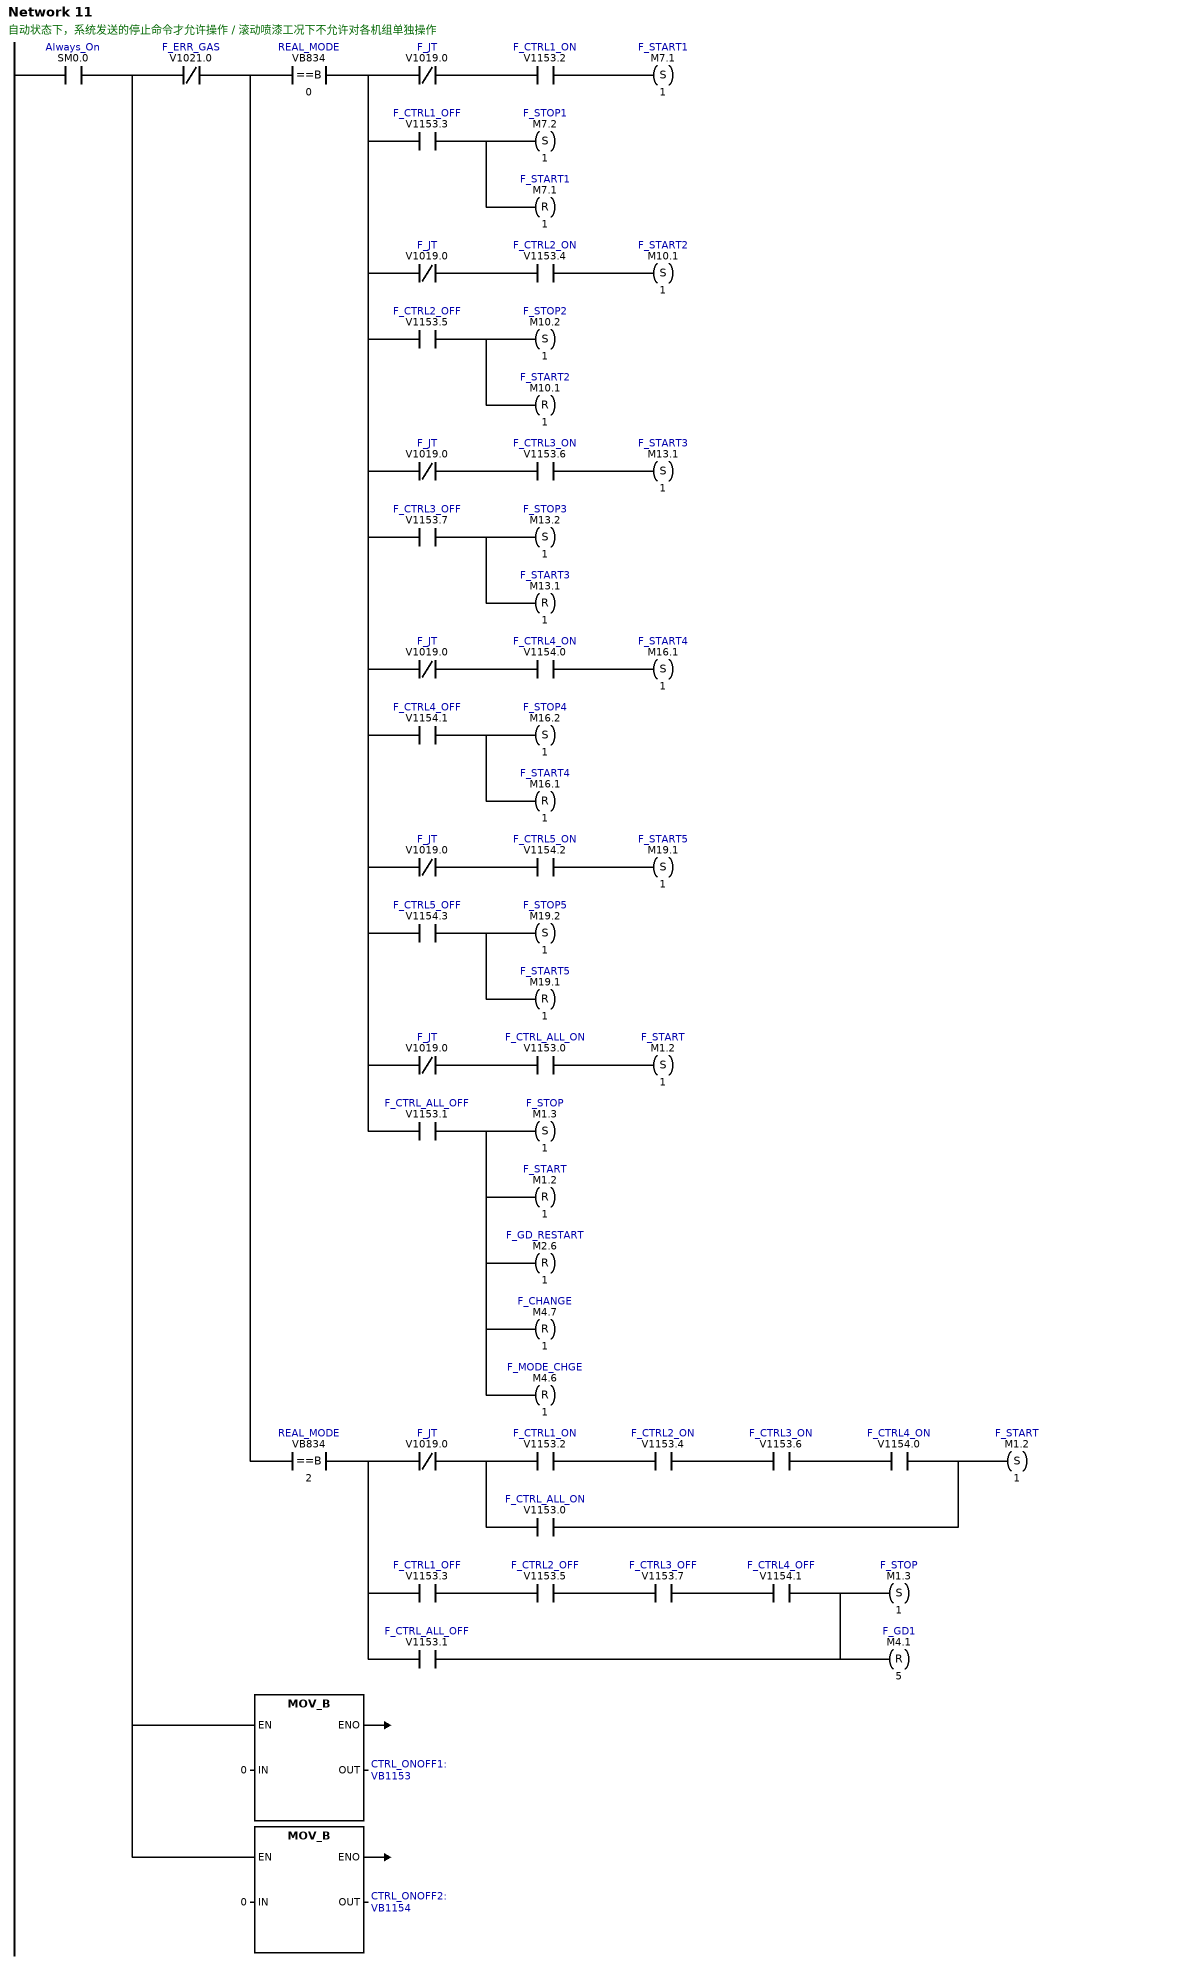
Network 11
// 自动状态下，系统发送的停止命令才允许操作
// 滚动喷漆工况下不允许对各机组单独操作
// (network saved uncompiled; LAD cells follow)
// row 0: c0 -| |- Always_On:SM0.0 v  c1 -|/|- F_ERR_GAS:V1021.0 v  c2 -|==B|- REAL_MODE:VB834, 0 v  c3 -|/|- F_JT:V1019.0  c4 -| |- F_CTRL1_ON:V1153.2  c5 -(S) F_START1:M7.1, 1
// row 1: c0 ^v  c1 ^v  c2 ^v  c3 -| |- F_CTRL1_OFF:V1153.3 v  c4 -(S) F_STOP1:M7.2, 1
// row 2: c0 ^v  c1 ^v  c2 ^v  c3 ^  c4 -(R) F_START1:M7.1, 1
// row 3: c0 ^v  c1 ^v  c2 ^v  c3 -|/|- F_JT:V1019.0  c4 -| |- F_CTRL2_ON:V1153.4  c5 -(S) F_START2:M10.1, 1
// row 4: c0 ^v  c1 ^v  c2 ^v  c3 -| |- F_CTRL2_OFF:V1153.5 v  c4 -(S) F_STOP2:M10.2, 1
// row 5: c0 ^v  c1 ^v  c2 ^v  c3 ^  c4 -(R) F_START2:M10.1, 1
// row 6: c0 ^v  c1 ^v  c2 ^v  c3 -|/|- F_JT:V1019.0  c4 -| |- F_CTRL3_ON:V1153.6  c5 -(S) F_START3:M13.1, 1
// row 7: c0 ^v  c1 ^v  c2 ^v  c3 -| |- F_CTRL3_OFF:V1153.7 v  c4 -(S) F_STOP3:M13.2, 1
// row 8: c0 ^v  c1 ^v  c2 ^v  c3 ^  c4 -(R) F_START3:M13.1, 1
// row 9: c0 ^v  c1 ^v  c2 ^v  c3 -|/|- F_JT:V1019.0  c4 -| |- F_CTRL4_ON:V1154.0  c5 -(S) F_START4:M16.1, 1
// row 10: c0 ^v  c1 ^v  c2 ^v  c3 -| |- F_CTRL4_OFF:V1154.1 v  c4 -(S) F_STOP4:M16.2, 1
// row 11: c0 ^v  c1 ^v  c2 ^v  c3 ^  c4 -(R) F_START4:M16.1, 1
// row 12: c0 ^v  c1 ^v  c2 ^v  c3 -|/|- F_JT:V1019.0  c4 -| |- F_CTRL5_ON:V1154.2  c5 -(S) F_START5:M19.1, 1
// row 13: c0 ^v  c1 ^v  c2 ^v  c3 -| |- F_CTRL5_OFF:V1154.3 v  c4 -(S) F_STOP5:M19.2, 1
// row 14: c0 ^v  c1 ^v  c2 ^v  c3 ^  c4 -(R) F_START5:M19.1, 1
// row 15: c0 ^v  c1 ^v  c2 ^v  c3 -|/|- F_JT:V1019.0  c4 -| |- F_CTRL_ALL_ON:V1153.0  c5 -(S) F_START:M1.2, 1
// row 16: c0 ^v  c1 ^v  c2 ^  c3 -| |- F_CTRL_ALL_OFF:V1153.1 v  c4 -(S) F_STOP:M1.3, 1
// row 17: c0 ^v  c1 ^v  c3 ^v  c4 -(R) F_START:M1.2, 1
// row 18: c0 ^v  c1 ^v  c3 ^v  c4 -(R) F_GD_RESTART:M2.6, 1
// row 19: c0 ^v  c1 ^v  c3 ^v  c4 -(R) F_CHANGE:M4.7, 1
// row 20: c0 ^v  c1 ^v  c3 ^  c4 -(R) F_MODE_CHGE:M4.6, 1
// row 21: c0 ^v  c1 ^  c2 -|==B|- REAL_MODE:VB834, 2 v  c3 -|/|- F_JT:V1019.0 v  c4 -| |- F_CTRL1_ON:V1153.2  c5 -| |- F_CTRL2_ON:V1153.4  c6 -| |- F_CTRL3_ON:V1153.6  c7 -| |- F_CTRL4_ON:V1154.0 v  c8 -(S) F_START:M1.2, 1
// row 22: c0 ^v  c2 ^v  c3 ^  c4 -| |- F_CTRL_ALL_ON:V1153.0  c5 --  c6 --  c7 -- ^
// row 23: c0 ^v  c2 ^v  c3 -| |- F_CTRL1_OFF:V1153.3  c4 -| |- F_CTRL2_OFF:V1153.5  c5 -| |- F_CTRL3_OFF:V1153.7  c6 -| |- F_CTRL4_OFF:V1154.1 v  c7 -(S) F_STOP:M1.3, 1
// row 24: c0 ^v  c2 ^  c3 -| |- F_CTRL_ALL_OFF:V1153.1  c4 --  c5 --  c6 -- ^  c7 -(R) F_GD1:M4.1, 5
// row 25: c0 ^v  c1 --  c2 [MOV_B EN:=power@row25, IN:=0, ENO=>power, OUT=>CTRL_ONOFF1:VB1153]  c3 ->
// row 26: c0 ^v  c2 [box]
// row 27: c0 ^  c1 --  c2 [MOV_B EN:=power@row27, IN:=0, ENO=>power, OUT=>CTRL_ONOFF2:VB1154]  c3 ->
// row 28: c2 [box]
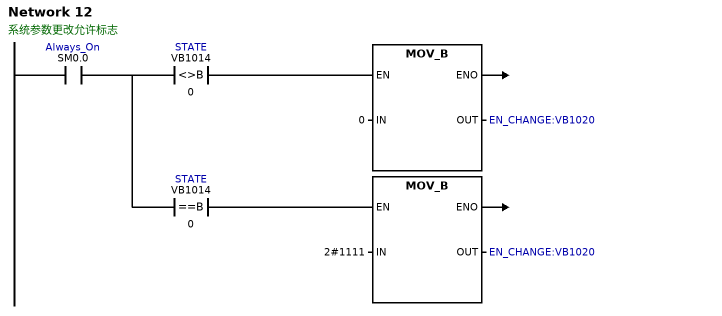
Network 12
// 系统参数更改允许标志
// (network saved uncompiled; LAD cells follow)
// row 0: c0 -| |- Always_On:SM0.0 v  c1 -|<>B|- STATE:VB1014, 0  c2 --  c3 [MOV_B EN:=power@row0, IN:=0, ENO=>power, OUT=>EN_CHANGE:VB1020]  c4 ->
// row 1: c0 ^v  c3 [box]
// row 2: c0 ^  c1 -|==B|- STATE:VB1014, 0  c2 --  c3 [MOV_B EN:=power@row2, IN:=2#1111, ENO=>power, OUT=>EN_CHANGE:VB1020]  c4 ->
// row 3: c3 [box]
END_SUBROUTINE_BLOCK

SUBROUTINE_BLOCK 参数设定:SBR5
TITLE=
VAR
TEMP_W:WORD;	// LW0 
TEMP_W1:WORD;	// LW2 
TEMP_W2:WORD;	// LW4 
END_VAR
BEGIN
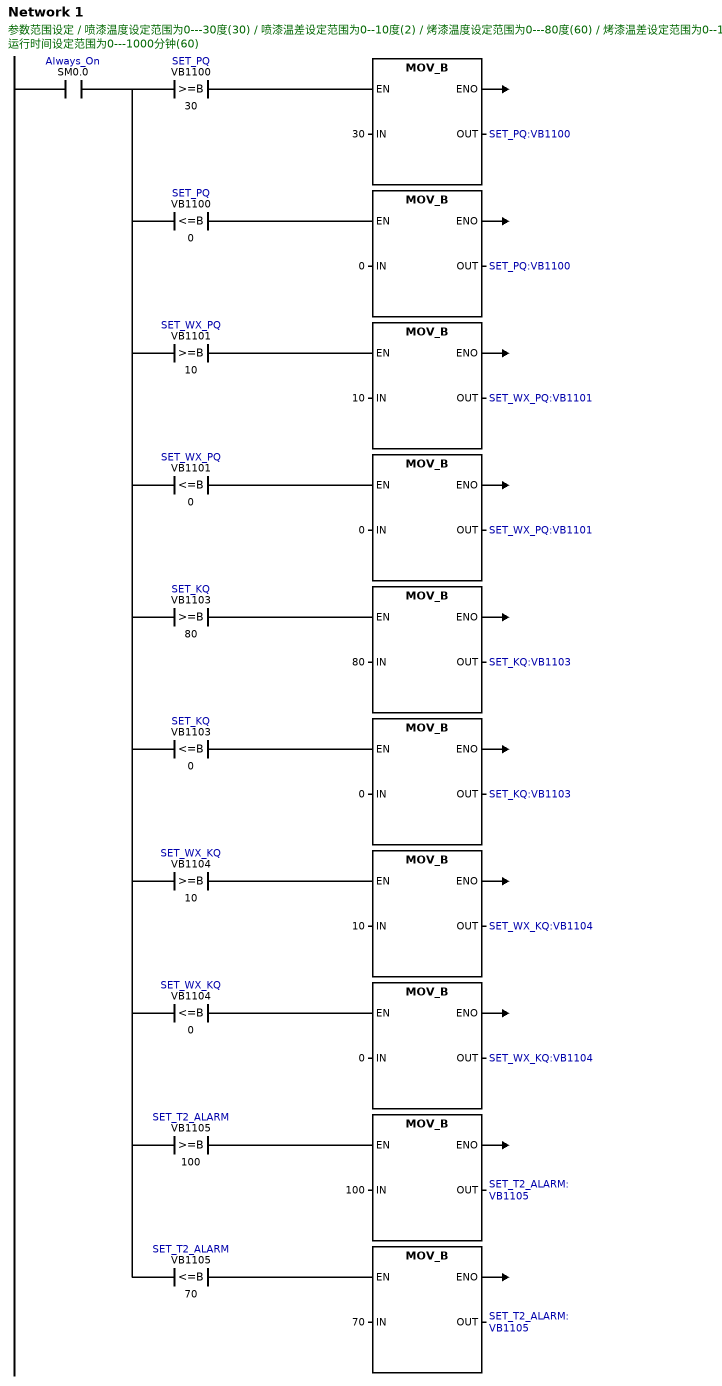
Network 1
// 参数范围设定
// 喷漆温度设定范围为0---30度(30)
// 喷漆温差设定范围为0--10度(2)
// 烤漆温度设定范围为0---80度(60)
// 烤漆温差设定范围为0--10度(2)
// T2超温保护温度设定范围为70---100度(85)
// 运行时间设定范围为0---1000分钟(60)
LD     Always_On:SM0.0
LPS
AB>=   SET_PQ:VB1100, 30
MOVB   30, SET_PQ:VB1100
LRD
AB<=   SET_PQ:VB1100, 0
MOVB   0, SET_PQ:VB1100
LRD
AB>=   SET_WX_PQ:VB1101, 10
MOVB   10, SET_WX_PQ:VB1101
LRD
AB<=   SET_WX_PQ:VB1101, 0
MOVB   0, SET_WX_PQ:VB1101
LRD
AB>=   SET_KQ:VB1103, 80
MOVB   80, SET_KQ:VB1103
LRD
AB<=   SET_KQ:VB1103, 0
MOVB   0, SET_KQ:VB1103
LRD
AB>=   SET_WX_KQ:VB1104, 10
MOVB   10, SET_WX_KQ:VB1104
LRD
AB<=   SET_WX_KQ:VB1104, 0
MOVB   0, SET_WX_KQ:VB1104
LRD
AB>=   SET_T2_ALARM:VB1105, 100
MOVB   100, SET_T2_ALARM:VB1105
LPP
AB<=   SET_T2_ALARM:VB1105, 70
MOVB   70, SET_T2_ALARM:VB1105
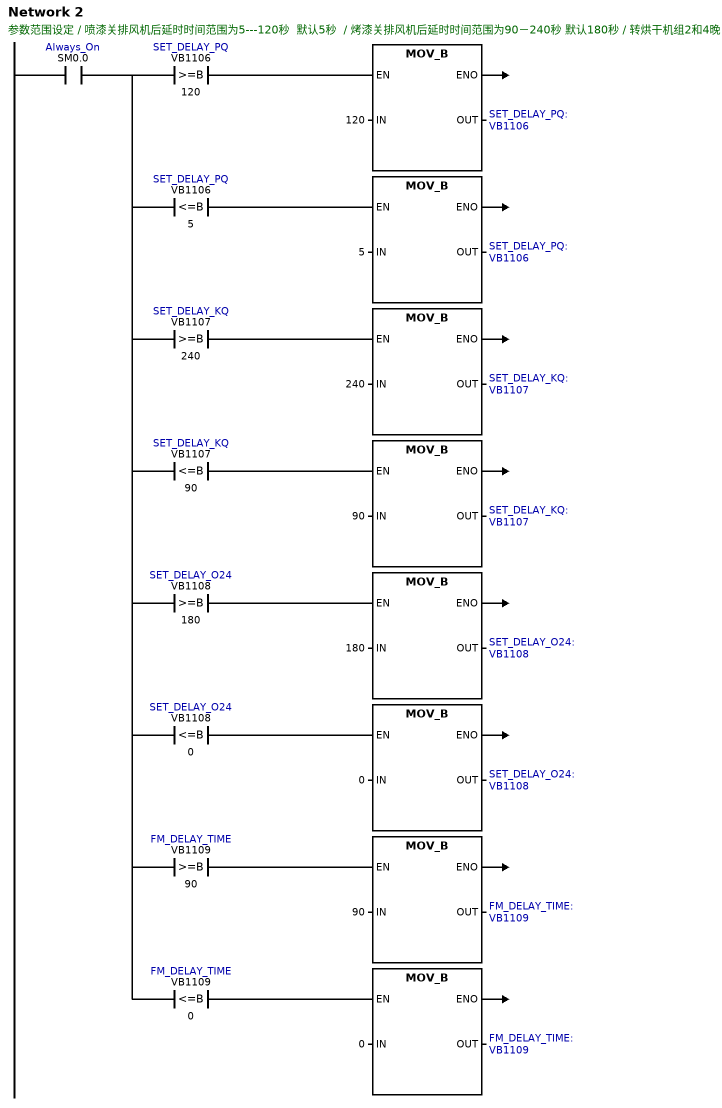
Network 2
// 参数范围设定
// 喷漆关排风机后延时时间范围为5---120秒  默认5秒 
// 烤漆关排风机后延时时间范围为90－240秒 默认180秒
// 转烘干机组2和4晚关延时时间为0－180秒   默认30秒
LD     Always_On:SM0.0
LPS
AB>=   SET_DELAY_PQ:VB1106, 120
MOVB   120, SET_DELAY_PQ:VB1106
LRD
AB<=   SET_DELAY_PQ:VB1106, 5
MOVB   5, SET_DELAY_PQ:VB1106
LRD
AB>=   SET_DELAY_KQ:VB1107, 240
MOVB   240, SET_DELAY_KQ:VB1107
LRD
AB<=   SET_DELAY_KQ:VB1107, 90
MOVB   90, SET_DELAY_KQ:VB1107
LRD
AB>=   SET_DELAY_O24:VB1108, 180
MOVB   180, SET_DELAY_O24:VB1108
LRD
AB<=   SET_DELAY_O24:VB1108, 0
MOVB   0, SET_DELAY_O24:VB1108
LRD
AB>=   FM_DELAY_TIME:VB1109, 90
MOVB   90, FM_DELAY_TIME:VB1109
LPP
AB<=   FM_DELAY_TIME:VB1109, 0
MOVB   0, FM_DELAY_TIME:VB1109
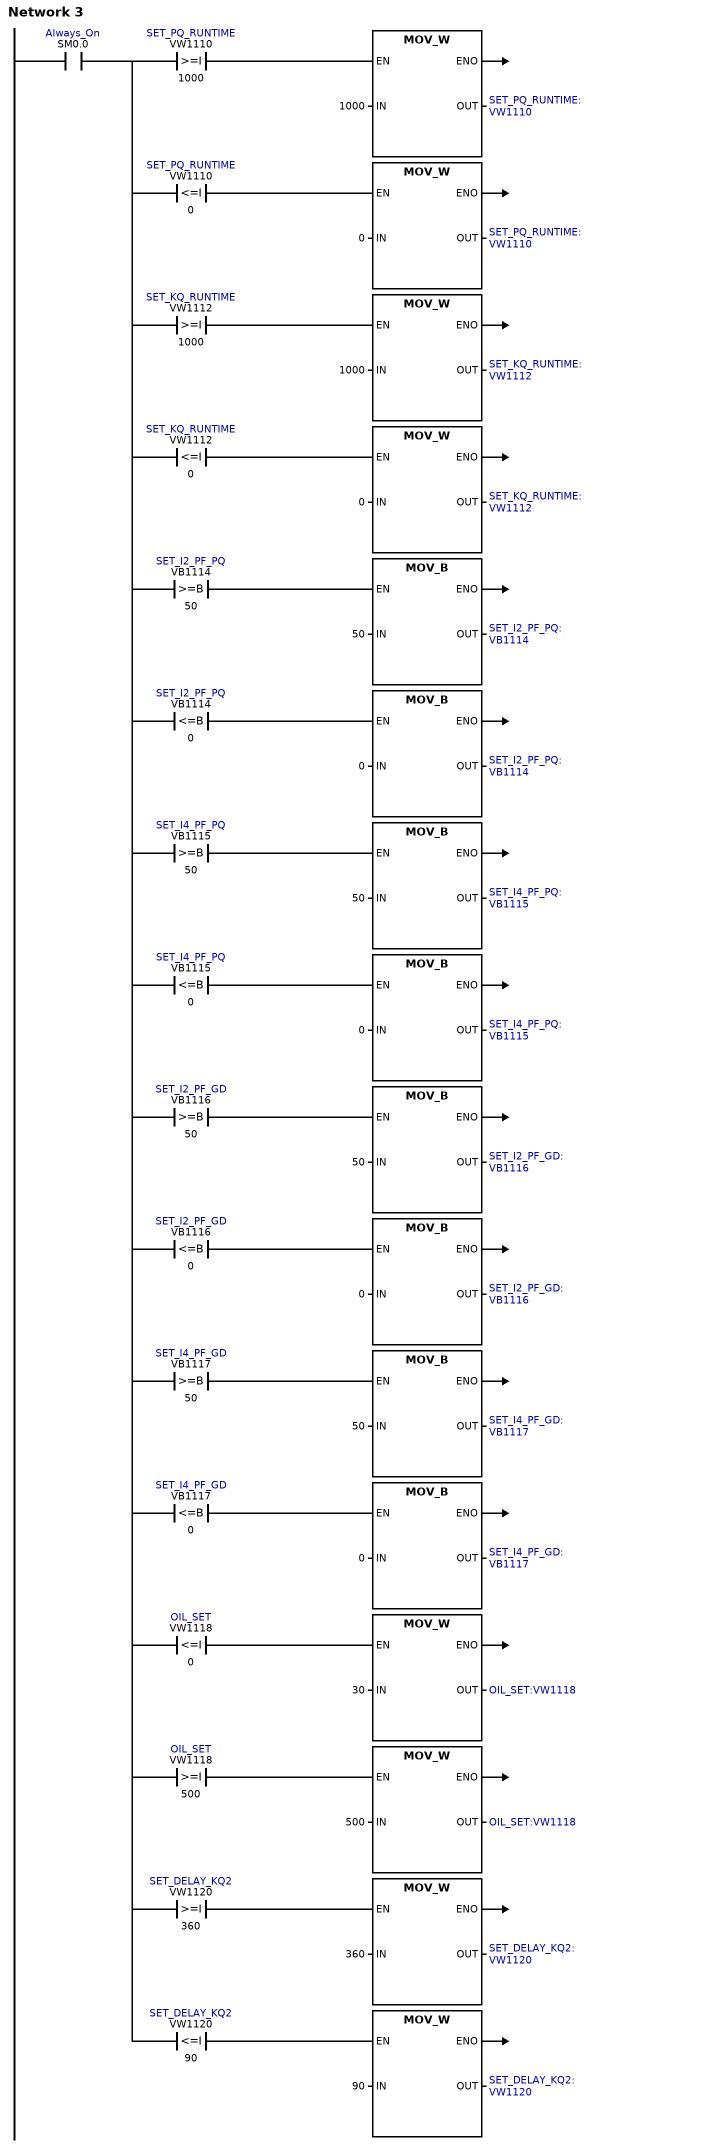
Network 3
LD     Always_On:SM0.0
LPS
AW>=   SET_PQ_RUNTIME:VW1110, 1000
MOVW   1000, SET_PQ_RUNTIME:VW1110
LRD
AW<=   SET_PQ_RUNTIME:VW1110, 0
MOVW   0, SET_PQ_RUNTIME:VW1110
LRD
AW>=   SET_KQ_RUNTIME:VW1112, 1000
MOVW   1000, SET_KQ_RUNTIME:VW1112
LRD
AW<=   SET_KQ_RUNTIME:VW1112, 0
MOVW   0, SET_KQ_RUNTIME:VW1112
LRD
AB>=   SET_I2_PF_PQ:VB1114, 50
MOVB   50, SET_I2_PF_PQ:VB1114
LRD
AB<=   SET_I2_PF_PQ:VB1114, 0
MOVB   0, SET_I2_PF_PQ:VB1114
LRD
AB>=   SET_I4_PF_PQ:VB1115, 50
MOVB   50, SET_I4_PF_PQ:VB1115
LRD
AB<=   SET_I4_PF_PQ:VB1115, 0
MOVB   0, SET_I4_PF_PQ:VB1115
LRD
AB>=   SET_I2_PF_GD:VB1116, 50
MOVB   50, SET_I2_PF_GD:VB1116
LRD
AB<=   SET_I2_PF_GD:VB1116, 0
MOVB   0, SET_I2_PF_GD:VB1116
LRD
AB>=   SET_I4_PF_GD:VB1117, 50
MOVB   50, SET_I4_PF_GD:VB1117
LRD
AB<=   SET_I4_PF_GD:VB1117, 0
MOVB   0, SET_I4_PF_GD:VB1117
LRD
AW<=   OIL_SET:VW1118, 0
MOVW   30, OIL_SET:VW1118
LRD
AW>=   OIL_SET:VW1118, 500
MOVW   500, OIL_SET:VW1118
LRD
AW>=   SET_DELAY_KQ2:VW1120, 360
MOVW   360, SET_DELAY_KQ2:VW1120
LPP
AW<=   SET_DELAY_KQ2:VW1120, 90
MOVW   90, SET_DELAY_KQ2:VW1120
